// TIA Portal project "LearningFactory_4_0_24V_V00" (V16)

(* hardware
DEVICE "ET 200SP-Station_1"  ET 200SP-Station
   slot 0: "Baugruppenträger_0"  Rack  6ES5 710-8MAx1
   slot 1: "PLC"  CPU 1512SP-1 PN  6ES7 512-1DK01-0AB0  V2.6
   slot 2: "DO1+2"  DQ 16x24VDC/0.5A ST  6ES7 132-6BH01-0BA0  V0.0
      slot 1: "DO1+2"  DQ 16x24VDC/0.5A ST
   slot 3: "DO3+4"  DQ 16x24VDC/0.5A ST  6ES7 132-6BH01-0BA0  V0.0
      slot 1: "DO3+4"  DQ 16x24VDC/0.5A ST
   slot 4: "DO5+6"  DQ 16x24VDC/0.5A ST  6ES7 132-6BH01-0BA0  V0.0
      slot 1: "DO5+6"  DQ 16x24VDC/0.5A ST
   slot 5: "DO7-14"  DQ 4x24VDC/2A HS  6ES7 132-6BD20-0DA0  V2.0
      slot 1: "DO7-14"  DQ 4x24VDC/2A HS
   slot 6: "DO15-22"  DQ 4x24VDC/2A HS  6ES7 132-6BD20-0DA0  V2.0
      slot 1: "DO15-22"  DQ 4x24VDC/2A HS
   slot 7: "DO23-30"  DQ 4x24VDC/2A HS  6ES7 132-6BD20-0DA0  V2.0
      slot 1: "DO23-30"  DQ 4x24VDC/2A HS
   slot 8: "DI1+2"  DI 16x24VDC ST  6ES7 131-6BH01-0BA0  V0.0
      slot 1: "DI1+2"  DI 16x24VDC ST
   slot 9: "DI3+4"  DI 16x24VDC ST  6ES7 131-6BH01-0BA0  V0.0
      slot 1: "DI3+4"  DI 16x24VDC ST
   slot 10: "DI5"  DI 8x24VDC HS  6ES7 131-6BF00-0DA0  V1.0
      slot 1: "DI5"  DI 8x24VDC HS
   slot 11: "DI6"  DI 8x24VDC HS  6ES7 131-6BF00-0DA0  V1.0
      slot 1: "DI6"  DI 8x24VDC HS
   slot 12: "AI7-10"  AI 2xU ST  6ES7 134-6FB00-0BA1  V1.0
      slot 1: "AI7-10"  AI 2xU ST
   slot 13: "End"  Server module  6ES7 193-6PA00-0AA0  V1.1
      slot 1: "End"  Server module
   slot 127: "BA 2xRJ45"  BA 2xRJ45  6ES7 193-6AR00-0AA0  V0.0
      slot 32769: "Port_1"  6ES7 193-6AR00-0AA0
      slot 32770: "Port_2"  6ES7 193-6AR00-0AA0
*)

// ===== PLC "PLC"  CPU 1512SP-1 PN =====

VAR_GLOBAL   // PLC tag table "VGR - Vacuum Gripper Robot"
   "IX_VGR_RefSwitchVerticalAxis_I1" AT %I1.6 : Bool;   // VGR - I1 = Reference switch vertical axis
   "IX_VGR_RefSwitchHorizontalAxis_I2" AT %I3.6 : Bool;   // VGR - I2 = Reference switch horizontal axis
   "IX_VGR_RefSwitchRotate_I3" AT %I3.7 : Bool;   // VGR - I3 = Reference switch rotate
   "IX_VGR_EncoderVerticalAxisImp1_B1" AT %I6.0 : Bool;   // VGR - B1 = Encoder vertical axis imulse 1
   "IX_VGR_EncoderVerticalAxisImp2_B2" AT %I6.4 : Bool;   // VGR - B2 = Encoder vertical axis imulse 2
   "IX_VGR_EncoderHorizontalAxisImp1_B3" AT %I6.1 : Bool;   // VGR - B3 = Encoder horizontal axis imulse 1
   "IX_VGR_EncoderHorizontalAxisImp2_B4" AT %I6.5 : Bool;   // VGR - B4 = Encoder horizontal axis imulse 2
   "IX_VGR_EncoderRotateImp1_B5" AT %I6.2 : Bool;   // VGR - B5 = Encoder rotate impulse 1
   "IX_VGR_EncoderRotateImp2_B6" AT %I6.6 : Bool;   // VGR - B6 = Encoder rotate impulse 2
   "QX_VGR_M1_VerticalAxisUp_Q1" AT %Q2.0 : Bool;   // VGR - Q1 = Motor M1 vertical axis up
   "QX_VGR_M1_VerticalAxisDown_Q2" AT %Q2.1 : Bool;   // VGR - Q2 = Motor M1 vertical axis down
   "QX_VGR_M2_HorizontalAxisBackward_Q3" AT %Q2.2 : Bool;   // VGR - Q3 = Motor M2 horizontal axis backward
   "QX_VGR_M2_HorizontalAxisForward_Q4" AT %Q2.3 : Bool;   // VGR - Q4 = Motor M2 horizontal axis forward
   "QX_VGR_M3_RotateClockwise_Q5" AT %Q2.4 : Bool;   // VGR - Q5 = Motor M3 rotate clockwise
   "QX_VGR_M3_RotateCounterclockwise_Q6" AT %Q2.5 : Bool;   // VGR - Q6 = Motor M3 rotate counterclockwise
   "QX_VGR_Compressor_Q7" AT %Q2.6 : Bool;   // VGR - Q7 = Compressor
   "QX_VGR_ValveVacuum_Q8" AT %Q2.7 : Bool;   // VGR - Q8 = Valve vacuum
   "QW_VGR_PWM_Vertical_M1" AT %QW15 : Int;   // VGR = PWM Motor M1 vertical axis
   "QW_VGR_PWM_Horizontal_M2" AT %QW17 : Int;   // VGR = PWM Motor M2 horizontal axis
   "QW_VGR_PWM_Rotate_M3" AT %QW19 : Int;   // VGR = PWM Motor M3 rotate axis
END_VAR

VAR_GLOBAL   // PLC tag table "HBW - Automated High-Bay Warehouse"
   "IX_HBW_RefSwitchHorizontalAxis_I1" AT %I1.0 : Bool;   // HBW - I1 = Reference switch horizontal axis
   "IX_HBW_LightBarrierInside_I2" AT %I1.1 : Bool;   // HBW - I2 = Light barrier inside
   "IX_HBW_LightBarrierOutside_I3" AT %I1.2 : Bool;   // HBW - I3 = Light barrier outside
   "IX_HBW_RefSwitchVerticalAxis_I4" AT %I1.3 : Bool;   // HBW - I4 = Reference switch vertical axis
   "IX_HBW_TrailSensor1Lower_A1" AT %I5.0 : Bool;   // HBW - A1 = Trail sensor (signal 1, lower)
   "IX_HBW_TrailSensor2Upper_A2" AT %I5.4 : Bool;   // HBW - A2 = Trail sensor (signal 2, upper)
   "IX_HBW_EncoderVerticalAxisImp1_B3" AT %I5.2 : Bool;   // HBW - B3 = Encoder vertical axis imulse 1
   "IX_HBW_EncoderVerticalAxisImp2_B4" AT %I5.6 : Bool;   // HBW - B4 = Encoder vertical axis imulse 2
   "IX_HBW_EncoderHorizontalAxisImp1_B1" AT %I5.1 : Bool;   // HBW - B1 = Encoder horizontal axis imulse 1
   "IX_HBW_EncoderHorizontalAxisImp2_B2" AT %I5.5 : Bool;   // HBW - B2 = Encoder horizontal axis imulse 2
   "IX_HBW_SwitchCantileverFront_I5" AT %I1.4 : Bool;   // HBW - I5 = Reference switch cantilever front
   "IX_HBW_SwitchCantileverBack_I6" AT %I1.5 : Bool;   // HBW - I6 = Reference switch cantilever back
   "QX_HBW_M1_ConveyorBeltForward_Q1" AT %Q1.0 : Bool;   // HBW - Q1 = Motor M1 conveyor belt forward
   "QX_HBW_M1_ConveyorBeltBackward_Q2" AT %Q1.1 : Bool;   // HBW - Q2 = Motor M1 conveyor belt backward
   "QX_HBW_M2_HorizontalTowardsRack_Q3" AT %Q1.2 : Bool;   // HBW - Q3 = Motor M2 horizontal towards rack
   "QX_HBW_M2_HorizontalTowardsConveyorBelt_Q4" AT %Q1.3 : Bool;   // HBW - Q4 = Motor M2 horizontal towards conveyor belt
   "QX_HBW_M3_VerticalAxisDownward_Q5" AT %Q1.4 : Bool;   // HBW - Q5 = Motor M3 vertical axis downward
   "QX_HBW_M3_VerticalAxisUpward_Q6" AT %Q1.5 : Bool;   // HBW - Q6 = Motor M3 vertical axis upward
   "QX_HBW_M4_CantileverForward_Q7" AT %Q1.6 : Bool;   // HBW - Q7 = Motor M4 cantilever forward
   "QX_HBW_M4_CantileverBackward_Q8" AT %Q1.7 : Bool;   // HBW - Q8 = Motor M4 cantilever backward
   "QW_HBW_PWM_ConveyorBelt_M1" AT %QW7 : Int;   // HBW = PWM Motor M1 conveyor belt
   "QW_HBW_PWM_HorizontalAxis_M2" AT %QW9 : Int;   // HBW = PWM Motor M2 horizontal axis
   "QW_HBW_PWM_VerticalAxis_M3" AT %QW11 : Int;   // HBW = PWM Motor M3 vertical axis
   "QW_HBW_PWM_Cantilever_M4" AT %QW13 : Int;   // HBW = PWM Motor M4 cantilever
END_VAR

VAR_GLOBAL   // PLC tag table "SLD - Sorting Line with Detection"
   "IX_SLD_PulseCounter_I1" AT %I3.0 : Bool;   // SLD - I1 = Pulse counter
   "IX_SLD_LightBarrierInlet_I2" AT %I3.1 : Bool;   // SLD - I2 = Light barrier inlet
   "IX_SLD_LightBarrierBehindColorSensor_I3" AT %I3.2 : Bool;   // SLD - I3 = Light barrier behind color sensor
   "IW_SLD_ColorSensor_A4" AT %IW7 : Word;   // SLD - A4 = Color sensor
   "IX_SLD_LightBarrierWhite_I5" AT %I3.3 : Bool;   // SLD - I5 = Light barrier white
   "IX_SLD_LightBarrierRed_I6" AT %I3.4 : Bool;   // SLD - I6 = Light barrier red
   "IX_SLD_LightBarrierBlue_I7" AT %I3.5 : Bool;   // SLD - I7 = Light barrier blue
   "QX_SLD_M1_ConveyorBelt_Q1" AT %Q5.0 : Bool;   // SLD - Q1 = Motor M1conveyor belt
   "QX_SLD_Compressor_Q2" AT %Q5.1 : Bool;   // SLD - Q2 = Compressor
   "QX_SLD_ValveFirstEjectorWhite_Q3" AT %Q5.2 : Bool;   // SLD - Q3 = Valve first ejector (white)
   "QX_SLD_ValveSecondEjectorRed_Q4" AT %Q5.3 : Bool;   // SLD - Q4 = Valve second ejector (red)
   "QX_SLD_ValveThirdEjectorBlue_Q5" AT %Q5.4 : Bool;   // SLD - Q5 = Valve third ejector (blue)
END_VAR

VAR_GLOBAL   // PLC tag table "MPO - Multi Processing Station with Oven"
   "IX_MPO_RefSwitchTurnTable_PosVac_I1" AT %I1.7 : Bool;   // MPO - I1 = Reference switch turn-table (position vacuum)
   "IX_MPO_RefSwitchTurnTable_PosBelt_I2" AT %I2.0 : Bool;   // MPO - I2 = Reference switch turn-table (position belt)
   "IX_MPO_LightBarrierEndOfConBelt_I3" AT %I2.1 : Bool;   // MPO - I3 = Light barrier end of conveyor belt
   "IX_MPO_RefSwitchTurnTable_PosSaw_I4" AT %I2.2 : Bool;   // MPO - I4 = Reference switch turn-table (position saw)
   "IX_MPO_RefSwitchVac_PosTurnTable_I5" AT %I2.3 : Bool;   // MPO - I5 = Reference switch vacuum (position turn-table)
   "IX_MPO_RefSwitchOvenFeederInside_I6" AT %I2.4 : Bool;   // MPO - I6 = Reference switch oven feeder inside
   "IX_MPO_RefSwitchOvenFeederOutside_I7" AT %I2.5 : Bool;   // MPO - I7 = Reference switch oven feeder outside
   "IX_MPO_RefSwitchVac_PosOven_I8" AT %I2.6 : Bool;   // MPO - I8 = Reference switch vacuum (position oven)
   "IX_MPO_LightBarrierOven_I9" AT %I2.7 : Bool;   // MPO - I9 = Light barrier oven
   "QX_MPO_M1_TurnTableClockwise_Q1" AT %Q3.0 : Bool;   // MPO - Q1 = Motor M1 turn-table clockwise
   "QX_MPO_M1_TurnTableCounterclockwise_Q2" AT %Q3.1 : Bool;   // MPO - Q2 = Motor M1 turn-table counterclockwise
   "QX_MPO_M2_ConveyorBeltForward_Q3" AT %Q3.2 : Bool;   // MPO - Q3 = Motor M2 conveyor belt forward
   "QX_MPO_M3_Saw_Q4" AT %Q3.3 : Bool;   // MPO - Q4 = Motor M3 saw
   "QX_MPO_M4_OvenFeederRetract_Q5" AT %Q3.4 : Bool;   // MPO - Q5 = Motor M4 oven feeder retract
   "QX_MPO_M4_OvenFeederExtend_Q6" AT %Q3.5 : Bool;   // MPO - Q6 = Motor M4 oven feeder extend
   "QX_MPO_M5_VacuumTowardsOven_Q7" AT %Q3.6 : Bool;   // MPO - Q7 = Motor M5 vacuum towards oven
   "QX_MPO_M5_VacuumTowardsTurnTable_Q8" AT %Q3.7 : Bool;   // MPO - Q8 = Motor M5 vacuum towards turn-table
   "QX_MPO_LightOven_Q9" AT %Q4.0 : Bool;   // MPO - Q9 = Light oven
   "QX_MPO_Compressor_Q10" AT %Q4.1 : Bool;   // MPO - Q10 = Compressor
   "QX_MPO_ValveVacuum_Q11" AT %Q4.2 : Bool;   // MPO - Q11 = Valve vacuum
   "QX_MPO_ValveLowering_Q12" AT %Q4.3 : Bool;   // MPO - Q12 = Valve lowering
   "QX_MPO_ValveOvenDoor_Q13" AT %Q4.4 : Bool;   // MPO - Q13 = Valve oven door
   "QX_MPO_ValveFeeder_Q14" AT %Q4.5 : Bool;   // MPO - Q14 = Valve feeder
   "QW_MPO_PWM_TurnTable_M1" AT %QW23 : Int;   // MPO = PWM Motor M1 turn-table
   "QW_MPO_PWM_Vacuum_M5" AT %QW25 : Int;   // MPO = PWM Motor M5 turn-table
END_VAR

VAR_GLOBAL   // PLC tag table "SSC - Sensor-Station Camera"
   "IX_SSC_RefSwitchVerticalAxis_I1" AT %I4.0 : Bool;   // SSC - ?? = Reference switch vertical axis / SSC - I1 = Reference switch vertical axis
   "IX_SSC_RefSwitchHorizontalAxis_I2" AT %I4.1 : Bool;   // SSC - ?? = Reference switch horizontal axis / SSC - I2 = Reference switch horizontal axis
   "IX_SSC_LightBarrierStorage_I3" AT %I4.3 : Bool;   // SSC - ?? = Light barrier inlet / SSC - I3 = Light barrier inlet
   "IX_SSC_LightBarrierOutsourcing_I4" AT %I4.2 : Bool;   // SSC - ?? = Light barrier behind color sensor / SSC - I4 = Light barrier behind color sensor
   "IW_SSC_ColorSensor_A1" AT %IW9 : Word;   // SSC - ?? = Color sensor / SSC - A1 = Color sensor
   "IX_SSC_EncoderVerticalAxisImp1_B1" AT %I5.3 : Bool;   // SSC - ?? = Encoder vertical axis imulse 1 / SSC - B1 = Encoder vertical axis imulse 1
   "IX_SSC_EncoderVerticalAxisImp2_B2" AT %I5.7 : Bool;   // SSC - ?? = Encoder vertical axis imulse 2 / SSC - B2 = Encoder vertical axis imulse 2
   "IX_SSC_EncoderHorizontalAxisImp1_B3" AT %I6.3 : Bool;   // SSC - ?? = Encoder horizontal axis imulse 1 / SSC - B3 = Encoder horizontal axis imulse 1
   "IX_SSC_EncoderHorizontalAxisImp2_B4" AT %I6.7 : Bool;   // SSC - ?? = Encoder horizontal axis imulse 2 / SSC - B4 = Encoder horizontal axis imulse 2
   "QX_SSC_M1_VerticalAxisUp_Q1" AT %Q6.0 : Bool;   // SSC - ?? = Motor M1 vertical axis up / SSC - Q1 = Motor M1 vertical axis up
   "QX_SSC_M1_VerticalAxisDown_Q2" AT %Q6.1 : Bool;   // SSC - ?? = Motor M1 vertical axis down / SSC - Q2 = Motor M1 vertical axis down
   "QX_SSC_M2_HorizontalAxisClockwise_Q3" AT %Q6.3 : Bool;   // SSC - ?? = Motor M2 horizontal axis backward / SSC - Q3 = Motor M2 horizontal axis backward
   "QX_SSC_M2_HorizontalAxisCounterclockwise_Q4" AT %Q6.2 : Bool;   // SSC - ?? = Motor M2 horizontal axis forward / SSC - Q4 = Motor M2 horizontal axis forward
   "QX_SSC_LED_Green_Q5" AT %Q6.4 : Bool;   // SSC - ?? = / SSC - Q5 = LED Green
   "QX_SSC_LED_Yellow_Q6" AT %Q6.5 : Bool;   // SSC - ?? = / SSC - Q6 = LED Yellow
   "QX_SSC_LED_Red_Q7" AT %Q6.6 : Bool;   // SSC - ?? = / SSC - Q7 = LED Red
   "QX_SSC_LED_Red_Online_Q8" AT %Q6.7 : Bool;   // SSC - ?? = / SSC - Q8 = LED Red Online
   "QW_SSC_PWM_Vertical_M1" AT %QW27 : Int;   // SSC - ?? = / SSC = PWM Motor M1 vertical axis
   "QW_SSC_PWM_Horizontal_M2" AT %QW29 : Int;   // SSC - ?? = / SSC = PWM Motor M2 horizontal axis
END_VAR

TYPE "typ_VGR"
   STRUCT
      x_NFC_Start_First : Bool;
      x_NFC_Start : Bool;
      x_NFC_Completed : Bool;
      x_HBW_Storage : Bool;
      x_HBW_Outsource : Bool;
      s_HBW_Outsource_Typ : String;
      x_HBW_Discards : Bool;
      x_HBW_PickedUp : Bool;
      x_MPO_Req_Discard : Bool;
      x_MPO_Discards : Bool;
      x_Ready_For_Outsource : Bool;
      x_State_Process : Bool;
      x_Workpiece_NiO : Bool;
      horizontal_Axis : "typ_Axis";
      vertical_Axis : "typ_Axis";
      rotate_Axis : "typ_Axis";
      Workpiece : "typ_Workpiece";
      History : Array[1..20] of "typ_History";
      di_Pos_DSI_horizontal : DInt;
      di_Pos_DSI_Collect_vertical : DInt;
      di_Pos_DSI_Discard_vertical : DInt;
      di_Offset_Pos_DSI_NFC_vertical : DInt;
      di_Pos_DSI_rotate : DInt;
      di_Pos_DSO_horizontal : DInt;
      di_Pos_DSO_Collect_vertical : DInt;
      di_Pos_DSO_Discard_vertical : DInt;
      di_Offset_Pos_DSO_vertical : DInt;
      di_Pos_DSO_rotate : DInt;
      di_Pos_Color_horizontal : DInt;
      di_Pos_Color_vertical : DInt;
      di_Pos_Color_rotate : DInt;
      di_Pos_NFC_horizontal : DInt;
      di_Pos_NFC_vertical : DInt;
      di_Pos_NFC_rotate : DInt;
      di_Pos_MPO_horizontal : DInt;
      di_Pos_MPO_vertical : DInt;
      di_Offset_Pos_MPO_vertical : DInt;
      di_Pos_MPO_rotate : DInt;
      di_Pos_HBW_horizontal : DInt;
      di_Offset_Pos_HBW_horizontal : DInt;
      di_Pos_HBW_Collect_vertical : DInt;
      di_Pos_HBW_Discard_vertical : DInt;
      di_Offset_Pos_HBW_vertical : DInt;
      di_Pos_HBW_rotate : DInt;
      di_Pos_NiO_horizontal : DInt;
      di_Pos_NiO_vertical : DInt;
      di_Pos_NiO_rotate : DInt;
      di_Pos_SLD_Blue_horizontal : DInt;
      di_Pos_SLD_Blue_vertical : DInt;
      di_Pos_SLD_Blue_rotate : DInt;
      di_Pos_SLD_Red_horizontal : DInt;
      di_Pos_SLD_Red_vertical : DInt;
      di_Pos_SLD_Red_rotate : DInt;
      di_Pos_SLD_White_horizontal : DInt;
      di_Pos_SLD_White_vertical : DInt;
      di_Pos_SLD_White_rotate : DInt;
   END_STRUCT;
END_TYPE

TYPE "typ_SetupAxis"
   STRUCT
      x_Setup_Activ : Bool;   // Einrichten Kalibrieren aktiv / Set up calibration active
      i_AxisSelection : Int;   // Nummer der Achse / Number of the axis
      i_Function : Int;   // 0= Automatic, 10=Ref. Fahrt, 20= Tippen, 30=Tippen mit Schritweite, 40= Pos. Anfahren / 0 = automatic, 10 = ref. Travel, 20 = tap, 30 = tap with step width, 40 = start
      x_Set_Ref_Pos : Bool;   // Referenzwert setzen / Set reference value
      x_Set_Soft_End_Pos : Bool;   // Softwareendlagen setzen / Set software end positions
      x_Approach_Ref_Pos : Bool;   // Referenz anfahren / Approach reference
      x_Axis_Pos : Bool;   // Achse positiv / Axis positiv
      x_Axis_Neg : Bool;   // Achse negativ / Axis negative
      x_Approach_Target_Pos : Bool;   // Zielposition anfahren / Approach Target position
      w_Increment : Word;   // Inkremente pro Schritt / Increments per step
      i_PWM : Int;   // PWM Signal
      di_Target_Position : DInt;   // Zielposition / Target position
      di_ActualPosition : DInt;   // Aktuelle Position / Actual position
      di_Ref_Pos : DInt;   // Referenzposition / Reference position
      di_Actual_Ref_Pos : DInt;   // Aktuelle Referenzposition / Current reference position
      di_Soft_End_Pos_Neg : DInt;   // Softwareendlage negativ / Software end position negative
      di_Actual_Soft_End_Pos_Neg : DInt;   // Aktuelle Softwareendlage negativ / Current software end position negative
      di_Soft_End_Pos_Pos : DInt;   // Softwareendlage positiv / Software end position positiv
      di_Actual_Soft_End_Pos_Pos : DInt;   // Aktuelle Softwareendlage positiv / Current software end position positiv
      di_LoopValue : DInt;   // Schleifenwert / Loop value
   END_STRUCT;
END_TYPE

TYPE "typ_Axis_Data"
   STRUCT
      di_Pos_Soft_Switch : DInt := 0;
      di_Neg_Soft_Switch : DInt := 0;
      di_Ref_Pos : DInt := 0;
      di_Loop_Value : DInt := 0;
      di_Pos_Window : DInt := 15;
   END_STRUCT;
END_TYPE

TYPE "typ_Axis"
   STRUCT
      x_Start_Positioning : Bool;
      x_Reference : Bool;
      x_Referenced : Bool;
      x_Position_Reached : Bool;
      di_Target_Position : DInt;
      di_Increment : DInt;
      di_Actual_Position : DInt := 0;
      i_PWM : Int;
      Config : "typ_Axis_Data";
   END_STRUCT;
END_TYPE

TYPE "typ_SSC"
   STRUCT
      x_Error : Bool;
      di_Pos_Centre_Horizontal : DInt;
      di_Pos_Centre_Vertical : DInt;
      di_Pos_HBW_Horizontal : DInt;
      di_Pos_HBW_Vertical : DInt;
      w_Threshold_White_Red : Word;
      w_Threshold_Red_Blue : Word;
      Horizontal_Axis : "typ_Axis";
      Vertical_Axis : "typ_Axis";
      Workpiece : "typ_Workpiece";
      History : Array[1..20] of "typ_History";
   END_STRUCT;
END_TYPE

TYPE "typ_HBW"
   STRUCT
      x_HBW_PickedUp_Accepted : Bool;
      x_HBW_Discards_Accepted : Bool;
      x_HBW_PickUp_Ready : Bool;
      x_HBW_Container_Available : Bool;
      x_Error : Bool;
      di_PosBelt_Horizontal : DInt;
      di_PosBelt_Vertical : DInt;
      di_Offset_Pos_Belt_Vertical : DInt;
      di_PosRack_A1_Horizontal : DInt;
      di_PosRack_A1_Vertical : DInt;
      di_PosRack_B2_Horizontal : DInt;
      di_PosRack_B2_Vertical : DInt;
      di_PosRack_C3_Horizontal : DInt;
      di_PosRack_C3_Vertical : DInt;
      di_Offset_Pos_Rack_Vertical : DInt;
      i_PWM_ConveyorBelt : Int := 800;
      i_PWM_Cantilever : Int := 800;
      Workpiece : "typ_Workpiece";
      History : Array[1..20] of "typ_History";
      Rack_Pos : Array[1..3, 1..3] of "typ_Rack_Pos";
      Rack_Workpiece : Array[1..3, 1..3] of "typ_Workpiece";
      Rack_History : Array[1..3, 1..3] of "typ_Rack_History";
      Horizontal_Axis : "typ_Axis";
      Vertical_Axis : "typ_Axis";
   END_STRUCT;
END_TYPE

TYPE "typ_Rack_Pos"
   STRUCT
      di_PosRack_Horizontal : DInt;
      di_PosRack_Vertical : DInt;
   END_STRUCT;
END_TYPE

TYPE "typ_MPO"
   STRUCT
      x_Discard_Ready : Bool;
      x_MPO_Discards_Accepted : Bool;
      x_Error : Bool;
      i_PWM_TurnTable : Int := 700;
      i_PWM_Vacuum : Int := 1000;
      Workpiece : "typ_Workpiece";
      History : Array[1..20] of "typ_History";
   END_STRUCT;
END_TYPE

TYPE "typ_SLD"
   STRUCT
      x_Error : Bool;
      i_CounterValue_Blue : Int := 8;
      i_CounterValue_White : Int := 2;
      i_CounterValue_Red : Int := 4;
      i_Counter_Actual : Int;
      w_Threshold_White_Red : Word;
      w_Threshold_Red_Blue : Word;
      Workpiece : "typ_Workpiece";
      History : Array[1..20] of "typ_History";
   END_STRUCT;
END_TYPE

TYPE "typ_Setup"
   STRUCT
      x_Clean_Rack_HBW : Bool;
      x_AcknowledgeButton : Bool;
      x_Color_Sensor_Calibration : Bool;
      x_Set_Calib_Value_Color_Blue : Bool;
      x_Set_Calib_Value_Color_White : Bool;
      x_Set_Calib_Value_Color_Red : Bool;
      x_Calculate_Value_Color : Bool;
      i_Color_Sensor_Selection : Int;
      w_Calib_ColorValue_Blue : Word;
      w_Calib_ColorValue_White : Word;
      w_Calib_ColorValue_Red : Word;
      w_Threshold_White_Red : Word;
      w_Threshold_Red_Blue : Word;
      w_Actual_ColorValue : Word;
      x_Set_Pos_Activ : Bool;   // Einrichten Kalibrieren aktiv / Set up calibration active
      x_Start_Positioning : Bool;
      x_Final_Positioning : Bool;
      x_Home_Positioning : Bool;
      x_Start_Offset : Bool;
      i_Pos_Selection : Int;   // Nummer der Achse / Number of the axis
      di_Pos_Horizontal : DInt;
      di_Pos_Vertical : DInt;
      di_Pos_Rotate : DInt;
      x_Counter_Value_Calibration : Bool;   // Einrichten Kalibrieren aktiv
      i_Calib_CounterValue_Blue : Int := 26;
      i_Calib_CounterValue_White : Int := 5;
      i_Calib_CounterValue_Red : Int := 16;
      x_Set_CounterValues : Bool;   // Einrichten Kalibrieren aktiv
      x_Activate_Continuous_Operation : Bool;
   END_STRUCT;
END_TYPE

TYPE "typ_Rack_History"
   STRUCT
      History : Array[1..20] of "typ_History";
   END_STRUCT;
END_TYPE

// folder: Dashboard types

TYPE "typ_Stock_Item"
   STRUCT
      ldt_ts : LDT;
      StockItem : Array[1..3, 1..3] of "typ_Workpiece";
      s_location : String;
   END_STRUCT;
END_TYPE

TYPE "typ_Acknowledgment_Client"
   STRUCT
      ldt_ts : LDT;
      i_code : Int;
      Workpiece : "typ_Workpiece";
   END_STRUCT;
END_TYPE

TYPE "typ_State_Client"
   STRUCT
      ldt_ts : LDT;
      s_station : String;
      i_code : Int;
      s_description : String;
      x_active : Bool;
      s_target : String;
   END_STRUCT;
END_TYPE

TYPE "typ_Broadcast"
   STRUCT
      ldt_ts : LDT;
      di_hardwareId : DInt;
      di_hardwareModel : DInt;
      s_softwareName : String;
      di_softwareVersion : DInt;
      s_message : String;
   END_STRUCT;
END_TYPE

TYPE "typ_Config_Camera_Picture"
   STRUCT
      ldt_ts : LDT;
      di_period : DInt;
   END_STRUCT;
END_TYPE

TYPE "typ_Config_Brightness_Sensor"
   STRUCT
      ldt_ts : LDT;
      x_on : Bool;
      i_fps : Int;
   END_STRUCT;
END_TYPE

TYPE "typ_Config_Enviorment_Sensor"
   STRUCT
      ldt_ts : LDT;
      di_period : DInt;
   END_STRUCT;
END_TYPE

TYPE "typ_History"
   STRUCT
      ldt_ts : LDT;
      i_code : Int;
   END_STRUCT;
END_TYPE

TYPE "typ_Pos_Pan_Tilt_Unit_Mov"
   STRUCT
      ldt_ts : LDT;
      s_cmd : String;
      i_degree : Int;
   END_STRUCT;
END_TYPE

TYPE "typ_Workpiece"
   STRUCT
      s_id : String;
      s_type : String;
      s_state : String;
   END_STRUCT;
END_TYPE

TYPE "typ_Order_Workpiece_Buttons_State"
   STRUCT
      ldt_ts : LDT;
      s_state : String;
      s_type : String;
   END_STRUCT;
END_TYPE

TYPE "typ_NFC_Module_State"
   STRUCT
      ldt_ts : LDT;
      Workpiece : "typ_Workpiece";
      History : Array[1..20] of "typ_History";
   END_STRUCT;
END_TYPE

TYPE "typ_VGR_Trigger"
   STRUCT
      ldt_ts : LDT;
      i_code : Int;
      Workpiece : "typ_Workpiece";
   END_STRUCT;
END_TYPE

TYPE "typ_Alert_Message"
   STRUCT
      ldt_ts : LDT;
      s_id : String;
      s_data : String;
      i_code : Int;
   END_STRUCT;
END_TYPE

TYPE "typ_Camera_Picture"
   STRUCT
      ldt_ts : LDT;
      s_data : String;
   END_STRUCT;
END_TYPE

TYPE "typ_Pos_Pan_Tilt_Unit_Enc"
   STRUCT
      ldt_ts : LDT;
      r_pan : Real;
      r_tilt : Real;
   END_STRUCT;
END_TYPE

TYPE "typ_Brightness_Sensor"
   STRUCT
      ldt_ts : LDT;
      r_br : Real;
      i_ldr : Int;
   END_STRUCT;
END_TYPE

TYPE "typ_Environment_Sensor"
   STRUCT
      ldt_ts : LDT;
      r_t : Real;
      r_rt : Real;
      r_h : Real;
      r_rh : Real;
      r_p : Real;
      i_iaq : Int;
      i_aq : Int;
      di_gr : DInt;
   END_STRUCT;
END_TYPE

TYPE "typ_Order_Workpiece_Buttons"
   STRUCT
      ldt_ts : LDT;
      s_type : String;
   END_STRUCT;
END_TYPE

TYPE "typ_Action_Buttons_NFC_Module"
   STRUCT
      ldt_ts : LDT;
      s_cmd : String;
   END_STRUCT;
END_TYPE

TYPE "typ_Joysticks"
   STRUCT
      ldt_ts : LDT;
      r_br : Real;
      i_ldr : Int;
   END_STRUCT;
END_TYPE

// folder: Interface Dashboard

TYPE "typ_MQTT_Interface_Dashboard"
   STRUCT
      Subscribe : "typ_MQTT_Interface_Dashboard_Subscribe";
      Publish : "typ_MQTT_ Interface_Dashboard_Publish";
   END_STRUCT;
END_TYPE

TYPE "typ_MQTT_ Interface_Dashboard_Publish"
   STRUCT
      ldt_AcknowledgeButton : LDT;
      ConfigRateEnviormentSensor : "typ_Config_Enviorment_Sensor";
      ConfigRateBrightnessSensor : "typ_Config_Brightness_Sensor";
      ConfigRateCameraPicture : "typ_Config_Camera_Picture";
      PosPanTiltUnit : "typ_Pos_Pan_Tilt_Unit_Mov";
      OrderWorkpieceButton : "typ_Order_Workpiece_Buttons";
      ActionButtonNFCModule : "typ_Action_Buttons_NFC_Module";
   END_STRUCT;
END_TYPE

TYPE "typ_MQTT_Interface_Dashboard_Subscribe"
   STRUCT
      EnvironmentSensor : "typ_Environment_Sensor";
      BrightnessSensor : "typ_Brightness_Sensor";
      CameraPicture : "typ_Camera_Picture";
      PosPanTiltUnit : "typ_Pos_Pan_Tilt_Unit_Enc";
      AlertMessage : "typ_Alert_Message";
      Broadcast : "typ_Broadcast";
      State_HBW : "typ_State_Client";
      State_VGR : "typ_State_Client";
      State_MPO : "typ_State_Client";
      State_SLD : "typ_State_Client";
      State_DSI : "typ_State_Client";
      State_DSO : "typ_State_Client";
      Stock_HBW : "typ_Stock_Item";
      State_Order : "typ_Order_Workpiece_Buttons_State";
      State_NFC_Device : "typ_NFC_Module_State";
   END_STRUCT;
END_TYPE

// folder: Interface TXT Controller

TYPE "typ_MQTT_Interface_TXT_Controller"
   STRUCT
      Subscribe : "typ_MQTT_Interface_TXT_Controler_Subscribe";
      Publish : "typ_MQTT_ Interface_TXT_Controler_Publish";
   END_STRUCT;
END_TYPE

TYPE "typ_MQTT_ Interface_TXT_Controler_Publish"
   STRUCT
      ActionButtonNFCModule : "typ_SPS_Action_Buttons_NFC_Module";
   END_STRUCT;
END_TYPE

TYPE "typ_MQTT_Interface_TXT_Controler_Subscribe"
   STRUCT
      State_NFC_Device : "typ_SPS_NFC_Module_State";
   END_STRUCT;
END_TYPE

// folder: TXT Controler Types

TYPE "typ_SPS_NFC_Module_State"
   STRUCT
      ldt_ts : LDT;
      Workpiece : "typ_Workpiece";
      History : Array[1..20] of "typ_History";
   END_STRUCT;
END_TYPE

TYPE "typ_SPS_Action_Buttons_NFC_Module"
   STRUCT
      ldt_ts : LDT;
      s_cmd : String;
      Workpiece : "typ_Workpiece";
      History : Array[1..20] of "typ_History";
   END_STRUCT;
END_TYPE

// folder: 2. Cloud

DATA_BLOCK "PRG_NFC_DB"   // DB12
{ S7_Optimized_Access := 'TRUE' }
VERSION : 0.1
// stored: InstanceOfName PRG_NFC
"PRG_NFC"
BEGIN
END_DATA_BLOCK

DATA_BLOCK "PRG_Acknowledge_DB"   // DB21
{ S7_Optimized_Access := 'TRUE' }
VERSION : 0.1
// stored: InstanceOfName PRG_Acknowledge
"PRG_Acknowledge"
BEGIN
END_DATA_BLOCK

DATA_BLOCK "PRG_Order_DB"   // DB25
{ S7_Optimized_Access := 'TRUE' }
VERSION : 0.1
// stored: InstanceOfName PRG_Order
"PRG_Order"
BEGIN
END_DATA_BLOCK

// folder: 3.1. VGR

DATA_BLOCK "PRG_VGR_Axis_horizontal_DB"   // DB8
{ S7_Optimized_Access := 'TRUE' }
VERSION : 0.1
// stored: InstanceOfName PRG_VGR_Axis_horizontal
"PRG_VGR_Axis_horizontal"
BEGIN
END_DATA_BLOCK

DATA_BLOCK "PRG_VGR_Axis_vertical_DB"   // DB9
{ S7_Optimized_Access := 'TRUE' }
VERSION : 0.1
// stored: InstanceOfName PRG_VGR_Axis_vertical
"PRG_VGR_Axis_vertical"
BEGIN
END_DATA_BLOCK

DATA_BLOCK "PRG_VGR_Axis_rotate_DB"   // DB10
{ S7_Optimized_Access := 'TRUE' }
VERSION : 0.1
// stored: InstanceOfName PRG_VGR_Axis_rotate
"PRG_VGR_Axis_rotate"
BEGIN
END_DATA_BLOCK

DATA_BLOCK "PRG_VGR_Axis_horizontal_Act_Pos_DB"   // DB15
{ S7_Optimized_Access := 'TRUE' }
VERSION : 0.1
// stored: InstanceOfName PRG_VGR_Axis_horizontal_Act_Pos
"PRG_VGR_Axis_horizontal_Act_Pos"
BEGIN
END_DATA_BLOCK

DATA_BLOCK "PRG_VGR_Ablauf_DB"   // DB19
{ S7_Optimized_Access := 'TRUE' }
VERSION : 0.1
// stored: InstanceOfName PRG_VGR_Ablauf
"PRG_VGR_Ablauf"
BEGIN
END_DATA_BLOCK

DATA_BLOCK "PRG_VGR_Axis_vertical_Act_Pos_DB"   // DB29
{ S7_Optimized_Access := 'TRUE' }
VERSION : 0.1
// stored: InstanceOfName PRG_VGR_Axis_vertical_Act_Pos
"PRG_VGR_Axis_vertical_Act_Pos"
BEGIN
END_DATA_BLOCK

DATA_BLOCK "PRG_VGR_Axis_rotate_Act_Pos_DB"   // DB31
{ S7_Optimized_Access := 'TRUE' }
VERSION : 0.1
// stored: InstanceOfName PRG_VGR_Axis_rotate_Act_Pos
"PRG_VGR_Axis_rotate_Act_Pos"
BEGIN
END_DATA_BLOCK

DATA_BLOCK "PRG_VGR_Set_Positioning_DB"   // DB34
{ S7_Optimized_Access := 'TRUE' }
VERSION : 0.1
// stored: InstanceOfName PRG_VGR_Set_Positioning
"PRG_VGR_Set_Positioning"
BEGIN
END_DATA_BLOCK

// folder: 3.2. HBW

DATA_BLOCK "PRG_HBW_Axis_Vertical_DB"   // DB14
{ S7_Optimized_Access := 'TRUE' }
VERSION : 0.1
// stored: InstanceOfName PRG_HBW_Axis_Vertical
"PRG_HBW_Axis_Vertical"
BEGIN
END_DATA_BLOCK

DATA_BLOCK "PRG_HBW_Axis_Horizontal_DB"   // DB18
{ S7_Optimized_Access := 'TRUE' }
VERSION : 0.1
// stored: InstanceOfName PRG_HBW_Axis_Horizontal
"PRG_HBW_Axis_Horizontal"
BEGIN
END_DATA_BLOCK

DATA_BLOCK "PRG_HBW_Ablauf_DB"   // DB22
{ S7_Optimized_Access := 'TRUE' }
VERSION : 0.1
// stored: InstanceOfName PRG_HBW_Ablauf
"PRG_HBW_Ablauf"
BEGIN
END_DATA_BLOCK

DATA_BLOCK "PRG_HBW_Axis_Horizontal_Act_Pos_DB"   // DB27
{ S7_Optimized_Access := 'TRUE' }
VERSION : 0.1
// stored: InstanceOfName PRG_HBW_Axis_Horizontal_Act_Pos
"PRG_HBW_Axis_Horizontal_Act_Pos"
BEGIN
END_DATA_BLOCK

DATA_BLOCK "PRG_HBW_Axis_Vertical_Act_Pos_DB"   // DB28
{ S7_Optimized_Access := 'TRUE' }
VERSION : 0.1
// stored: InstanceOfName PRG_HBW_Axis_Vertical_Act_Pos
"PRG_HBW_Axis_Vertical_Act_Pos"
BEGIN
END_DATA_BLOCK

DATA_BLOCK "PRG_HBW_Set_Positioning_DB"   // DB35
{ S7_Optimized_Access := 'TRUE' }
VERSION : 0.1
// stored: InstanceOfName PRG_HBW_Set_Positioning
"PRG_HBW_Set_Positioning"
BEGIN
END_DATA_BLOCK

// folder: 3.3. MPO

DATA_BLOCK "PRG_MPO_Ablauf_DB"   // DB5
{ S7_Optimized_Access := 'TRUE' }
VERSION : 0.1
// stored: InstanceOfName PRG_MPO_Ablauf
"PRG_MPO_Ablauf"
BEGIN
END_DATA_BLOCK

// folder: 3.4. SLD

DATA_BLOCK "PRG_SLD_Ablauf_DB"   // DB20
{ S7_Optimized_Access := 'TRUE' }
VERSION : 0.1
// stored: InstanceOfName PRG_SLD_Ablauf
"PRG_SLD_Ablauf"
BEGIN
END_DATA_BLOCK

DATA_BLOCK "PRG_SLD_Calibration_Color_DB"   // DB38
{ S7_Optimized_Access := 'TRUE' }
VERSION : 0.1
// stored: InstanceOfName PRG_SLD_Calibration_Color
"PRG_SLD_Calibration_Color"
BEGIN
END_DATA_BLOCK

DATA_BLOCK "PRG_SLD_Set_Counter_Values_DB"   // DB39
{ S7_Optimized_Access := 'TRUE' }
VERSION : 0.1
// stored: InstanceOfName PRG_SLD_Set_Counter_Values
"PRG_SLD_Set_Counter_Values"
BEGIN
END_DATA_BLOCK

// folder: 3.5. SSC

DATA_BLOCK "PRG_SSC_Axis_Vertical_DB"   // DB3
{ S7_Optimized_Access := 'TRUE' }
VERSION : 0.1
// stored: InstanceOfName PRG_SSC_Axis_Vertical
"PRG_SSC_Axis_Vertical"
BEGIN
END_DATA_BLOCK

DATA_BLOCK "PRG_SSC_Axis_Vertical_Act_Pos_DB"   // DB6
{ S7_Optimized_Access := 'TRUE' }
VERSION : 0.1
// stored: InstanceOfName PRG_SSC_Axis_Vertical_Act_Pos
"PRG_SSC_Axis_Vertical_Act_Pos"
BEGIN
END_DATA_BLOCK

DATA_BLOCK "PRG_SSC_Axis_Horizontal_DB"   // DB7
{ S7_Optimized_Access := 'TRUE' }
VERSION : 0.1
// stored: InstanceOfName PRG_SSC_Axis_Horizontal
"PRG_SSC_Axis_Horizontal"
BEGIN
END_DATA_BLOCK

DATA_BLOCK "PRG_SSC_Ablauf_DB"   // DB16
{ S7_Optimized_Access := 'TRUE' }
VERSION : 0.1
// stored: InstanceOfName PRG_SSC_Ablauf
"PRG_SSC_Ablauf"
BEGIN
END_DATA_BLOCK

DATA_BLOCK "PRG_SSC_Light_DB"   // DB26
{ S7_Optimized_Access := 'TRUE' }
VERSION : 0.1
// stored: InstanceOfName PRG_SSC_Light
"PRG_SSC_Light"
BEGIN
END_DATA_BLOCK

DATA_BLOCK "PRG_SSC_Axis_Horizontal_Act_Pos_DB"   // DB30
{ S7_Optimized_Access := 'TRUE' }
VERSION : 0.1
// stored: InstanceOfName PRG_SSC_Axis_Horizontal_Act_Pos
"PRG_SSC_Axis_Horizontal_Act_Pos"
BEGIN
END_DATA_BLOCK

DATA_BLOCK "PRG_DSI_Status_DB"   // DB32
{ S7_Optimized_Access := 'TRUE' }
VERSION : 0.1
// stored: InstanceOfName PRG_DSI_Status
"PRG_DSI_Status"
BEGIN
END_DATA_BLOCK

DATA_BLOCK "PRG_DSO_Status_DB"   // DB33
{ S7_Optimized_Access := 'TRUE' }
VERSION : 0.1
// stored: InstanceOfName PRG_DSO_Status
"PRG_DSO_Status"
BEGIN
END_DATA_BLOCK

DATA_BLOCK "PRG_SSC_Set_Positioning_DB"   // DB36
{ S7_Optimized_Access := 'TRUE' }
VERSION : 0.1
// stored: InstanceOfName PRG_SSC_Set_Positioning
"PRG_SSC_Set_Positioning"
BEGIN
END_DATA_BLOCK

DATA_BLOCK "PRG_SSC_Calibration_Color_DB"   // DB37
{ S7_Optimized_Access := 'TRUE' }
VERSION : 0.1
// stored: InstanceOfName PRG_SSC_Calibration_Color
"PRG_SSC_Calibration_Color"
BEGIN
END_DATA_BLOCK

// folder: 4. Global Declaration

DATA_BLOCK "gtyp_Interface_Dashboard"   // DB1
TITLE = Global Interface Dashboard Cloud
{ S7_Optimized_Access := 'TRUE' }
AUTHOR : A.Schaefer
VERSION : 0.0
BEGIN
END_DATA_BLOCK

DATA_BLOCK "gtyp_VGR"   // DB2
TITLE = Global DB VGR
{ S7_Optimized_Access := 'TRUE' }
AUTHOR : A.Schaefer
VERSION : 0.0
BEGIN
   di_Pos_DSI_Collect_vertical := 2950;
   di_Pos_MPO_vertical := 1800;
   di_Pos_HBW_Discard_vertical := 200;
   vertical_Axis.Config.di_Pos_Soft_Switch := 20000;
   horizontal_Axis.Config.di_Pos_Soft_Switch := 20000;
   rotate_Axis.Config.di_Pos_Soft_Switch := 20000;
   di_Pos_DSI_horizontal := 20;
   di_Pos_DSI_rotate := 30;
   di_Pos_Color_horizontal := 150;
   di_Pos_Color_rotate := 430;
   di_Pos_Color_vertical := 2450;
   di_Pos_NFC_vertical := 2450;
   di_Pos_NFC_horizontal := 900;
   di_Pos_NFC_rotate := 700;
   di_Pos_HBW_rotate := 5350;
   di_Offset_Pos_DSI_NFC_vertical := 1200;
   di_Offset_Pos_HBW_vertical := 100;
   di_Pos_HBW_horizontal := 600;
   di_Pos_SLD_Red_rotate := 1460;
   di_Pos_SLD_White_rotate := 1770;
   di_Pos_SLD_Blue_rotate := 1200;
   di_Pos_SLD_Red_vertical := 3100;
   di_Pos_SLD_White_vertical := 3100;
   di_Pos_SLD_Blue_vertical := 3100;
   di_Pos_SLD_Red_horizontal := 1580;
   di_Pos_SLD_White_horizontal := 1370;
   di_Pos_SLD_Blue_horizontal := 2150;
   di_Pos_DSO_rotate := 970;
   di_Pos_MPO_rotate := 3500;
   di_Pos_NiO_rotate := 1100;
   di_Pos_DSO_horizontal := 2070;
   di_Pos_DSO_Discard_vertical := 1480;
   di_Pos_NiO_vertical := 2700;
   di_Pos_MPO_horizontal := 3400;
   di_Pos_HBW_Collect_vertical := 650;
   di_Offset_Pos_MPO_vertical := 650;
   horizontal_Axis.i_PWM := 500;
   vertical_Axis.i_PWM := 500;
   rotate_Axis.i_PWM := 500;
   di_Offset_Pos_DSO_vertical := 500;
END_DATA_BLOCK

DATA_BLOCK "gtyp_SetupAxis"   // DB4
TITLE = Global DB Setup Axis
{ S7_Optimized_Access := 'TRUE' }
AUTHOR : A.Schaefer
VERSION : 0.0
BEGIN
END_DATA_BLOCK

DATA_BLOCK "gtyp_MPO"   // DB11
TITLE = Global DB MPO
{ S7_Optimized_Access := 'TRUE' }
AUTHOR : A.Schaefer
VERSION : 0.0
BEGIN
END_DATA_BLOCK

DATA_BLOCK "gtyp_SSC"   // DB13
TITLE = Global DB SSC
{ S7_Optimized_Access := 'TRUE' }
AUTHOR : A.Schaefer
VERSION : 0.0
BEGIN
   Horizontal_Axis.Config.di_Pos_Soft_Switch := 5450;
   Vertical_Axis.Config.di_Pos_Soft_Switch := 3000;
   di_Pos_Centre_Horizontal := 3000;
   di_Pos_Centre_Vertical := 1400;
   Vertical_Axis.Config.di_Pos_Window := 25;
   Horizontal_Axis.Config.di_Pos_Window := 25;
   di_Pos_HBW_Horizontal := 5400;
   di_Pos_HBW_Vertical := 950;
   Horizontal_Axis.i_PWM := 1000;
   Vertical_Axis.i_PWM := 1000;
   w_Threshold_White_Red := 16#25DA;
   w_Threshold_Red_Blue := 16#3C57;
END_DATA_BLOCK

DATA_BLOCK "gtyp_HBW"   // DB17
TITLE = Global DB HBW
{ S7_Optimized_Access := 'TRUE' }
AUTHOR : A.Schaefer
VERSION : 0.0
BEGIN
   Horizontal_Axis.Config.di_Pos_Soft_Switch := 7900;
   Vertical_Axis.Config.di_Pos_Soft_Switch := 3350;
   di_PosBelt_Vertical := 2800;
   di_PosBelt_Horizontal := 18;
   di_Offset_Pos_Belt_Vertical := 370;
   Rack_Pos[1,1].di_PosRack_Horizontal := 2870;
   Rack_Pos[1,1].di_PosRack_Vertical := 400;
   Rack_Pos[1,2].di_PosRack_Horizontal := 5200;
   Rack_Pos[1,2].di_PosRack_Vertical := 400;
   Rack_Pos[1,3].di_PosRack_Horizontal := 7550;
   Rack_Pos[1,3].di_PosRack_Vertical := 400;
   Rack_Pos[2,1].di_PosRack_Horizontal := 2870;
   Rack_Pos[2,2].di_PosRack_Horizontal := 5200;
   Rack_Pos[2,3].di_PosRack_Horizontal := 7550;
   Rack_Pos[2,1].di_PosRack_Vertical := 1750;
   Rack_Pos[2,2].di_PosRack_Vertical := 1750;
   Rack_Pos[2,3].di_PosRack_Vertical := 1750;
   Rack_Pos[3,1].di_PosRack_Horizontal := 2870;
   Rack_Pos[3,1].di_PosRack_Vertical := 3150;
   Rack_Pos[3,2].di_PosRack_Horizontal := 5200;
   Rack_Pos[3,2].di_PosRack_Vertical := 3150;
   Rack_Pos[3,3].di_PosRack_Horizontal := 7550;
   Rack_Pos[3,3].di_PosRack_Vertical := 3150;
   Horizontal_Axis.Config.di_Pos_Window := 15;
   Vertical_Axis.Config.di_Pos_Window := 15;
   Horizontal_Axis.i_PWM := 700;
   Vertical_Axis.i_PWM := 600;
   Rack_Workpiece[1,1].s_id := '0';
   Rack_Workpiece[1,2].s_id := '0';
   Rack_Workpiece[1,3].s_id := '0';
   Rack_Workpiece[2,1].s_id := '0';
   Rack_Workpiece[2,2].s_id := '0';
   Rack_Workpiece[2,3].s_id := '0';
   Rack_Workpiece[3,1].s_id := '0';
   Rack_Workpiece[3,2].s_id := '0';
   Rack_Workpiece[3,3].s_id := '0';
   di_PosRack_A1_Horizontal := 2870;
   di_PosRack_A1_Vertical := 400;
   di_PosRack_B2_Horizontal := 5200;
   di_PosRack_B2_Vertical := 1750;
   di_PosRack_C3_Horizontal := 7560;
   di_PosRack_C3_Vertical := 3250;
   di_Offset_Pos_Rack_Vertical := 370;
   i_PWM_Cantilever := 1000;
END_DATA_BLOCK

DATA_BLOCK "gtyp_Setup"   // DB23
TITLE = Global DB Setup
{ S7_Optimized_Access := 'TRUE' }
AUTHOR : A.Schaefer
VERSION : 0.0
BEGIN
END_DATA_BLOCK

DATA_BLOCK "gtyp_SLD"   // DB24
TITLE = Global DB SLD
{ S7_Optimized_Access := 'TRUE' }
AUTHOR : A.Schaefer
VERSION : 0.0
BEGIN
   i_CounterValue_White := 5;
   i_CounterValue_Blue := 26;
   i_CounterValue_Red := 16;
   w_Threshold_White_Red := 16#2698;
   w_Threshold_Red_Blue := 16#3D41;
END_DATA_BLOCK

DATA_BLOCK "gtyp_Interface_TXT_Controler"   // DB40
{ S7_Optimized_Access := 'TRUE' }
VERSION : 0.1
BEGIN
END_DATA_BLOCK

DATA_BLOCK "RT_INFO_scl_OB30"   // DB325
{ S7_Optimized_Access := 'TRUE' }
VERSION : 0.1
   VAR
      mode : UInt := 1;   // Mode 1 = Runtime of a specific OB; 2 = Maximum runtime of a specific OB; 3 = Minimum runtime of a specific OB; 10 = Mean value of the percentage of total runtime used by higher-priority OBs; ...
      obNbr : OB_Any := 1;   // OB to read
      infoData : LTime;   // mode 1 --> Runtime in LTIME
      returnValue : Int;   // Error information of instruction
   END_VAR
BEGIN
END_DATA_BLOCK

DATA_BLOCK "RT_INFO_scl_OB1"   // DB326
{ S7_Optimized_Access := 'TRUE' }
VERSION : 0.1
   VAR
      mode : UInt := 1;   // Mode 1 = Runtime of a specific OB; 2 = Maximum runtime of a specific OB; 3 = Minimum runtime of a specific OB; 10 = Mean value of the percentage of total runtime used by higher-priority OBs; ...
      obNbr : OB_Any := 1;   // OB to read
      infoData : LTime;   // mode 1 --> Runtime in LTIME
      returnValue : Int;   // Error information of instruction
   END_VAR
BEGIN
END_DATA_BLOCK

// folder: (top level)

ORGANIZATION_BLOCK "Main"   // OB1, SCL, ProgramCycle
TITLE = "Main Program Sweep (Cycle)"
{ S7_Optimized_Access := 'TRUE' }
AUTHOR : A.Schaefer
VERSION : 0.0
   VAR_INPUT
      Initial_Call : Bool;   // Initial call of this OB
      Remanence : Bool;   // =True, if remanent data are available
   END_VAR
BEGIN
   // current cycle Time OB30
   "RT_INFO_scl_OB30".mode := 1;
   "RT_INFO_scl_OB30".obNbr := 30;
   "RT_INFO_scl_OB30".returnValue := RT_INFO(MODE := "RT_INFO_scl_OB30".mode,
                                             OB := "RT_INFO_scl_OB30".obNbr,
                                             INFO := "RT_INFO_scl_OB30".infoData);

   // current cycle Time OB1
   "RT_INFO_scl_OB1".mode := 1;
   "RT_INFO_scl_OB1".obNbr := 1;
   "RT_INFO_scl_OB1".returnValue := RT_INFO(MODE := "RT_INFO_scl_OB1".mode,
                                            OB := "RT_INFO_scl_OB1".obNbr,
                                            INFO := "RT_INFO_scl_OB1".infoData);

   // sources SSC
   "PRG_SSC_Ablauf_DB"();
   "PRG_SSC_Set_Positioning_DB"();
   "PRG_SSC_Calibration_Color_DB"();
   "PRG_SSC_Axis_Vertical_DB"();
   "PRG_SSC_Axis_Horizontal_DB"();
   "PRG_SSC_Light_DB"();

   // sources VGR
   "PRG_VGR_Ablauf_DB"();
   "PRG_VGR_Set_Positioning_DB"();
   "PRG_VGR_Axis_horizontal_DB"();
   "PRG_VGR_Axis_vertical_DB"();
   "PRG_VGR_Axis_rotate_DB"();
   "PRG_NFC_DB"();

   // sources HBW
   "PRG_HBW_Ablauf_DB"();
   "PRG_HBW_Set_Positioning_DB"();
   "PRG_HBW_Axis_Vertical_DB"();
   "PRG_HBW_Axis_Horizontal_DB"();

   // sources MPO
   "PRG_MPO_Ablauf_DB"();

   // sources SLD
   "PRG_SLD_Ablauf_DB"();
   "PRG_SLD_Calibration_Color_DB"();
   "PRG_SLD_Set_Counter_Values_DB"();

   // sources input/output
   "PRG_DSI_Status_DB"();
   "PRG_DSO_Status_DB"();

   // sources dashboard
   "PRG_Order_DB"();
   "PRG_Acknowledge_DB"();
END_ORGANIZATION_BLOCK

ORGANIZATION_BLOCK "Cyclic interrupt"   // OB30, SCL, CyclicInterrupt
TITLE = Cyclic interrupt
{ S7_Optimized_Access := 'TRUE' }
AUTHOR : A.Schaefer
VERSION : 0.0
   VAR_INPUT
      Initial_Call : Bool;   // Initial call of this OB
      Event_Count : Int;   // Events discarded
   END_VAR
   VAR_TEMP
      li_Return_LDT : Int;
   END_VAR
BEGIN

   "PRG_SSC_Axis_Horizontal_Act_Pos_DB"();
   "PRG_SSC_Axis_Vertical_Act_Pos_DB"();

   "PRG_HBW_Axis_Horizontal_Act_Pos_DB"();
   "PRG_HBW_Axis_Vertical_Act_Pos_DB"();

   "PRG_VGR_Axis_horizontal_Act_Pos_DB"();
   "PRG_VGR_Axis_vertical_Act_Pos_DB"();
   "PRG_VGR_Axis_rotate_Act_Pos_DB"();
END_ORGANIZATION_BLOCK

// folder: 1. FB / FC

FUNCTION_BLOCK "FB_Blinker"   // FB2, SCL
TITLE = Functionblock Blinker
{ S7_Optimized_Access := 'TRUE' }
AUTHOR : A.Schaefer
VERSION : 0.0
   VAR_INPUT
      int_periodendauer : Time;
   END_VAR
   VAR_OUTPUT
      outx_blinker : Bool;
   END_VAR
   VAR
      lfb_ton : TON_TIME;
      lx_esv_timer : Bool;
      lx_blinker : Bool;
   END_VAR
BEGIN
   #lfb_ton(IN := NOT #lx_esv_timer,
           PT := #int_periodendauer / 2,
           Q => #lx_esv_timer);

   IF #lx_esv_timer THEN
       #lx_blinker := NOT #lx_blinker;
   END_IF;

   #outx_blinker := #lx_blinker;
END_FUNCTION_BLOCK

FUNCTION_BLOCK "FB_INC_DEC"   // FB9, SCL
TITLE = Funktionblock Increment decodition
{ S7_Optimized_Access := 'TRUE' }
AUTHOR : A.Schaefer
VERSION : 0.0
   VAR_INPUT
      inx_CHa : Bool := false;
      inx_CHb : Bool := false;
      inx_RST : Bool := False;
      ini_Ref_Wert : Int := 0;
   END_VAR
   VAR_OUTPUT
      outx_dir : Bool := false;
      outi_cnt : Int := 0;
   END_VAR
   VAR
      lx_edgea : Bool := False;
      lx_clka : Bool;
      lx_clkb : Bool;
      lx_edgeb : Bool;
      lx_axb : Bool;
      lx_dir : Bool;
      li_cnt : Int;
   END_VAR
BEGIN

   #lx_axb := #inx_CHa XOR #inx_CHb;

   (* create pulses for channel a *)
   #lx_clka := #inx_CHa XOR #lx_edgea;
   #lx_edgea := #inx_CHa;

   #lx_clkb := #inx_CHb XOR #lx_edgeb;
   #lx_edgeb := #inx_CHb;

   (* create pulses for both channels *)
   #lx_clka := #lx_clka OR #lx_clkb;

   (* set the direction output *)
   IF #lx_axb AND #lx_clka THEN
       #lx_dir := TRUE;
   END_IF;
   IF #lx_axb AND #lx_clkb THEN
       #lx_dir := FALSE;
   END_IF;

   (* increment or decrement the counter *)
   IF #lx_clka AND #lx_dir THEN
       #li_cnt := #li_cnt + 1;
   END_IF;
   IF #lx_clka AND NOT #lx_dir THEN
       #li_cnt := #li_cnt - 1;
   END_IF;

   (* reset the counter if rst active *)
   IF #inx_RST THEN
       #li_cnt := #ini_Ref_Wert;
   END_IF;

   #outx_dir := #lx_dir;
   #outi_cnt := #li_cnt;
END_FUNCTION_BLOCK

FUNCTION_BLOCK "FB_Axis"   // FB22, SCL
TITLE = Functionblock Axis
{ S7_Optimized_Access := 'TRUE' }
AUTHOR : A.Schaefer
VERSION : 0.0
   VAR_INPUT
      ini_Axis : Int;
      indi_Increment : DInt;
      inx_Ref_Switch : Bool;
      inx_Start_Positioning : Bool;
      inx_Referencing : Bool;
      ini_PWM : Int;
      indi_Target_Position : DInt;
   END_VAR
   VAR_OUTPUT
      outx_Referenced : Bool;
      outx_Position_Reached : Bool;
      outx_Motor_Pos : Bool;
      outx_Motor_Neg : Bool;
      outi_Motor_PWM : Int;
      outdi_Actual_Position : DInt;
   END_VAR
   VAR_IN_OUT
      inouttyp_Config : "typ_Axis_Data";
      inouttyp_Setup : "typ_SetupAxis";
   END_VAR
   VAR
      li_StepCaseSetup : Int;
      li_StepCase : Int;
      lx_Init : Bool;
      lx_Motor_Neg : Bool;
      lx_Motor_Pos : Bool;
      lx_Start_TON_Wait : Bool;
      li_PWM : Int;
      ldi_ValueStep : DInt;
      ldi_Actual_Position : DInt;
      ldi_Actual_Position_Old : DInt;
      lfb_R_Trig_Setup : R_TRIG;
      lfb_R_Trig_Referencing : R_TRIG;
      lfb_TON_Wait : TON_TIME;
   END_VAR
BEGIN
   IF #lx_Init THEN

       // rising edge set up axis
       #lfb_R_Trig_Setup(CLK := #inouttyp_Setup.x_Setup_Activ);

       //Reload when switching to set up
       IF #lfb_R_Trig_Setup.Q THEN
           #inouttyp_Setup.di_LoopValue               := #inouttyp_Config.di_Loop_Value;
           #inouttyp_Setup.di_Ref_Pos                 := 
           #inouttyp_Setup.di_Actual_Ref_Pos          := #inouttyp_Config.di_Ref_Pos;
           #inouttyp_Setup.di_Soft_End_Pos_Neg        := 
           #inouttyp_Setup.di_Actual_Soft_End_Pos_Neg := #inouttyp_Config.di_Neg_Soft_Switch;
           #inouttyp_Setup.di_Soft_End_Pos_Pos        :=
           #inouttyp_Setup.di_Actual_Soft_End_Pos_Pos := #inouttyp_Config.di_Pos_Soft_Switch;
           #inouttyp_Setup.i_PWM                      := #ini_PWM;
           #inouttyp_Setup.x_Approach_Ref_Pos         := FALSE;
           #inouttyp_Setup.x_Approach_Target_Pos      := FALSE;
           #inouttyp_Setup.x_Axis_Neg                 := FALSE;
           #inouttyp_Setup.x_Axis_Pos                 := FALSE;
           #inouttyp_Setup.x_Set_Ref_Pos              := FALSE;
           #inouttyp_Setup.x_Set_Soft_End_Pos         := FALSE;
       END_IF;

       #ldi_Actual_Position := #indi_Increment;

       //rising edge referencing
       #lfb_R_Trig_Referencing(CLK := #inx_Referencing);

       //waiting period
       #lfb_TON_Wait(IN := #lx_Start_TON_Wait,
                     PT := T#200ms);

       (**********************************)
       (******   set up step chain   *****)
       (**********************************)
       IF #inouttyp_Setup.i_AxisSelection = #ini_Axis AND #inouttyp_Setup.x_Setup_Activ THEN
           IF #inouttyp_Setup.x_Approach_Ref_Pos THEN
               #inouttyp_Setup.i_Function := 10;
           END_IF;

           CASE #inouttyp_Setup.i_Function OF

               0:  // automatic
                   #ldi_Actual_Position_Old := 0;
                   #inouttyp_Setup.x_Approach_Ref_Pos := FALSE;
                   #lx_Start_TON_Wait := FALSE;

               10: // homing
                   IF #inouttyp_Setup.x_Approach_Ref_Pos THEN
                       IF NOT #inx_Ref_Switch THEN
                           #lx_Motor_Neg := TRUE;
                           #lx_Motor_Pos := FALSE;
                           #outx_Referenced := FALSE;
                       END_IF;

                       IF #inx_Ref_Switch THEN
                           #lx_Motor_Neg := TRUE;
                           #lx_Motor_Pos := TRUE;

                           IF #ldi_Actual_Position = #inouttyp_Config.di_Ref_Pos THEN
                               #inouttyp_Setup.x_Approach_Ref_Pos := FALSE;
                               #lx_Motor_Neg       := FALSE;
                               #lx_Motor_Pos       := FALSE;
                               #outx_Referenced    := TRUE;
                           END_IF;
                       END_IF;
                   END_IF;

               20:  // tap
                   #lx_Motor_Neg := #inouttyp_Setup.x_Axis_Neg AND NOT #inx_Ref_Switch AND NOT (#ldi_Actual_Position <= #inouttyp_Setup.di_Soft_End_Pos_Neg);
                   #lx_Motor_Pos := #inouttyp_Setup.x_Axis_Pos AND NOT #lx_Motor_Neg AND NOT (#ldi_Actual_Position >= #inouttyp_Setup.di_Soft_End_Pos_Pos);

               30:  // tap with increment
                   #ldi_Actual_Position_Old := #ldi_Actual_Position;

                   // positiv
                   IF #inouttyp_Setup.x_Axis_Pos AND NOT ((#ldi_Actual_Position + #inouttyp_Setup.w_Increment + #inouttyp_Setup.di_LoopValue) >= #inouttyp_Setup.di_Soft_End_Pos_Pos) THEN
                       #lx_Motor_Neg := FALSE;
                       #lx_Motor_Pos := TRUE;
                       #ldi_ValueStep := #ldi_Actual_Position_Old + #inouttyp_Setup.w_Increment;

                       // without loop
                       IF (#inouttyp_Setup.di_LoopValue = 0) THEN
                           #inouttyp_Setup.i_Function := 36;
                       ELSE
                           #inouttyp_Setup.i_Function := 31;
                       END_IF;
                   // negativ
                   ELSIF #inouttyp_Setup.x_Axis_Neg AND NOT ((#ldi_Actual_Position - #inouttyp_Setup.w_Increment) <= #inouttyp_Config.di_Neg_Soft_Switch) THEN
                       #lx_Motor_Neg := TRUE;
                       #lx_Motor_Pos := FALSE;
                       #ldi_ValueStep := #ldi_Actual_Position_Old - #inouttyp_Setup.w_Increment;
                       #inouttyp_Setup.i_Function := 34;
                   END_IF;

               31: // with loop
                   IF ((#ldi_Actual_Position >= (#ldi_ValueStep + #inouttyp_Setup.di_LoopValue - #inouttyp_Config.di_Pos_Window)) = 0) THEN
                       #lx_Motor_Neg := TRUE;
                       #lx_Motor_Pos := TRUE;
                       #inouttyp_Setup.i_Function := 32;
                   END_IF;

               32: // wait sequence
                   #lx_Start_TON_Wait := TRUE;

                   IF #lfb_TON_Wait.Q THEN
                       #lx_Motor_Neg               := FALSE;
                       #lx_Motor_Pos               := FALSE;
                       #lx_Start_TON_Wait          := FALSE;
                       #inouttyp_Setup.i_Function  := 33;
                   END_IF;

               33: // change direction
                   #lx_Motor_Neg := TRUE;
                   #lx_Motor_Pos := FALSE;
                   #inouttyp_Setup.i_Function := 34;

               34: // position reached negativ
                   IF (#ldi_Actual_Position <= (#ldi_ValueStep + #inouttyp_Config.di_Pos_Window))
                       AND (#ldi_Actual_Position >= (#ldi_ValueStep - #inouttyp_Config.di_Pos_Window)) THEN
                       #lx_Motor_Neg := TRUE;
                       #lx_Motor_Pos := TRUE;
                       #inouttyp_Setup.i_Function := 35;
                   END_IF;

               35: // wait sequence
                   #lx_Start_TON_Wait := TRUE;

                   IF #lfb_TON_Wait.Q THEN
                       #lx_Motor_Neg := FALSE;
                       #lx_Motor_Pos := FALSE;
                       #lx_Start_TON_Wait := FALSE;
                       #inouttyp_Setup.x_Axis_Neg := FALSE;
                       #inouttyp_Setup.x_Axis_Pos := FALSE;
                       #inouttyp_Setup.i_Function := 30;
                   END_IF;


               36: // position reached positiv
                   IF (#ldi_Actual_Position <= (#ldi_ValueStep + #inouttyp_Config.di_Pos_Window))
                       AND (#ldi_Actual_Position >= (#ldi_ValueStep - #inouttyp_Config.di_Pos_Window)) THEN
                       #lx_Motor_Neg := TRUE;
                       #lx_Motor_Pos := TRUE;
                       #inouttyp_Setup.i_Function := 37;
                   END_IF;

               37: // wait sequence
                   #lx_Start_TON_Wait := TRUE;

                   IF #lfb_TON_Wait.Q THEN
                       #lx_Motor_Neg := FALSE;
                       #lx_Motor_Pos := FALSE;
                       #lx_Start_TON_Wait := FALSE;
                       #inouttyp_Setup.x_Axis_Neg := FALSE;
                       #inouttyp_Setup.x_Axis_Pos := FALSE;
                       #inouttyp_Setup.i_Function := 30;
                   END_IF;

               40: // approach position
                   IF #inouttyp_Setup.x_Approach_Target_Pos THEN
                       // positiv
                       IF (#inouttyp_Setup.di_Target_Position > #ldi_Actual_Position) AND NOT ((#inouttyp_Setup.di_Target_Position + #inouttyp_Setup.di_LoopValue) >= #inouttyp_Setup.di_Soft_End_Pos_Pos)  THEN
                           #lx_Motor_Neg := FALSE;
                           #lx_Motor_Pos := TRUE;
                           // without loop
                           IF (#inouttyp_Setup.di_LoopValue = 0) THEN
                               #inouttyp_Setup.i_Function := 46;
                           ELSE
                               #inouttyp_Setup.i_Function := 41;
                           END_IF;
                       // negativ
                       ELSIF ((#inouttyp_Setup.di_Target_Position < #ldi_Actual_Position) AND NOT (#inouttyp_Setup.di_Target_Position <= #inouttyp_Config.di_Neg_Soft_Switch))  THEN
                           #lx_Motor_Neg := TRUE;
                           #lx_Motor_Pos := FALSE;
                           #inouttyp_Setup.i_Function := 44;
                       ELSIF (#inouttyp_Setup.di_Target_Position = #ldi_Actual_Position) THEN
                           #inouttyp_Setup.i_Function := 46;
                       END_IF;

                   END_IF;

               41: // with loop
                   IF (#ldi_Actual_Position >= (#inouttyp_Setup.di_Target_Position + #inouttyp_Setup.di_LoopValue - #inouttyp_Config.di_Pos_Window)) THEN
                       #lx_Motor_Neg := TRUE;
                       #lx_Motor_Pos := TRUE;
                       #inouttyp_Setup.i_Function := 42;
                   END_IF;

               42: // wait sequence
                   #lx_Start_TON_Wait := TRUE;

                   IF #lfb_TON_Wait.Q THEN
                       #lx_Motor_Neg := FALSE;
                       #lx_Motor_Pos := FALSE;
                       #lx_Start_TON_Wait := FALSE;
                       #inouttyp_Setup.i_Function := 43;
                   END_IF;

               43: // change direction
                   #lx_Motor_Neg   := TRUE;
                   #lx_Motor_Pos   := FALSE;
                   #inouttyp_Setup.i_Function     := 44;

               44: // position reached negativ
                   IF (#ldi_Actual_Position <= (#inouttyp_Setup.di_Target_Position + #inouttyp_Config.di_Pos_Window))
                       AND (#ldi_Actual_Position >= (#inouttyp_Setup.di_Target_Position - #inouttyp_Config.di_Pos_Window)) THEN
                       #lx_Motor_Neg := TRUE;
                       #lx_Motor_Pos := TRUE;
                       #inouttyp_Setup.i_Function := 45;
                   END_IF;

               45: // wait sequence
                   #lx_Start_TON_Wait := TRUE;

                   IF #lfb_TON_Wait.Q THEN
                       #lx_Motor_Neg := FALSE;
                       #lx_Motor_Pos := FALSE;
                       #lx_Start_TON_Wait := FALSE;
                       #inouttyp_Setup.x_Axis_Neg := FALSE;
                       #inouttyp_Setup.x_Axis_Pos := FALSE;
                       #inouttyp_Setup.i_Function := 40;
                   END_IF;

               46: //  position reached positiv
                   IF (#ldi_Actual_Position <= (#inouttyp_Setup.di_Target_Position + #inouttyp_Config.di_Pos_Window))
                       AND (#ldi_Actual_Position >= (#inouttyp_Setup.di_Target_Position - #inouttyp_Config.di_Pos_Window)) THEN
                       #lx_Motor_Neg := TRUE;
                       #lx_Motor_Pos := TRUE;
                       #inouttyp_Setup.i_Function := 47;
                   END_IF;

               47:  // wait sequence
                   #lx_Start_TON_Wait := TRUE;

                   IF #lfb_TON_Wait.Q THEN
                       #lx_Motor_Neg := FALSE;
                       #lx_Motor_Pos := FALSE;
                       #lx_Start_TON_Wait := FALSE;
                       #inouttyp_Setup.x_Approach_Target_Pos := FALSE;
                       #inouttyp_Setup.i_Function := 40;
                   END_IF;
               ELSE  // Statement section ELSE
                   ;
           END_CASE;

           // set reference point
           IF #inouttyp_Setup.x_Set_Ref_Pos THEN
               #inouttyp_Setup.di_Actual_Ref_Pos   :=
               #inouttyp_Config.di_Ref_Pos         := #inouttyp_Setup.di_Ref_Pos;
               #inouttyp_Setup.x_Set_Ref_Pos       := FALSE;
           END_IF;

           // set software end position
           IF #inouttyp_Setup.x_Set_Soft_End_Pos THEN
               #inouttyp_Setup.di_Actual_Soft_End_Pos_Neg  :=
               #inouttyp_Config.di_Neg_Soft_Switch         := #inouttyp_Setup.di_Soft_End_Pos_Neg;
               #inouttyp_Setup.di_Actual_Soft_End_Pos_Pos  :=
               #inouttyp_Config.di_Pos_Soft_Switch         := #inouttyp_Setup.di_Soft_End_Pos_Pos;
               #inouttyp_Setup.x_Set_Soft_End_Pos := FALSE;
           END_IF;

           // reload PWM
           #li_PWM := #inouttyp_Setup.i_PWM;

           // reload actual position
           #inouttyp_Setup.di_ActualPosition           := #ldi_Actual_Position;

       (************************************)
       (******   position step chain   *****)
       (************************************)
       ELSIF NOT #inouttyp_Setup.x_Setup_Activ THEN

           // rising edge set up axis
           IF #lfb_R_Trig_Referencing.Q THEN
               #li_StepCase := 0;
           END_IF;

           CASE #li_StepCase OF

               0:  // init
                   #lx_Start_TON_Wait := FALSE;

                   IF #inx_Referencing THEN
                       #li_StepCase            := 10;
                       #outx_Position_Reached  := FALSE;
                       #outx_Referenced        := FALSE;
                   ELSIF #inx_Start_Positioning THEN
                       #li_StepCase            := 20;
                       #outx_Position_Reached  := FALSE;
                   END_IF;

               10: // homing
                   IF NOT #inx_Ref_Switch THEN
                       #lx_Motor_Neg := TRUE;
                       #lx_Motor_Pos := FALSE;
                   END_IF;

                   IF #inx_Ref_Switch THEN
                       #lx_Motor_Neg := TRUE;
                       #lx_Motor_Pos := TRUE;

                       IF #inx_Ref_Switch THEN
                           IF #ldi_Actual_Position = #inouttyp_Config.di_Ref_Pos THEN
                               #lx_Motor_Neg := FALSE;
                               #lx_Motor_Pos := FALSE;
                               #outx_Referenced := TRUE;
                               #li_StepCase := 11;
                           END_IF;
                       END_IF;
                   END_IF;

               11: // wait not referencing
                   IF NOT #inx_Referencing THEN
                       #li_StepCase := 0;
                   END_IF;

               20: // approach position
                   // positiv
                   IF (#indi_Target_Position > #ldi_Actual_Position) AND NOT ((#indi_Target_Position + #inouttyp_Config.di_Loop_Value) >= #inouttyp_Config.di_Pos_Soft_Switch) THEN
                       #lx_Motor_Neg := FALSE;
                       #lx_Motor_Pos := TRUE;
                       //without loop
                       IF (#inouttyp_Config.di_Loop_Value = 0) THEN
                           #li_StepCase := 26;
                       ELSE
                           #li_StepCase := 21;
                       END_IF;
                   // negativ
                   ELSIF ((#indi_Target_Position < #ldi_Actual_Position) AND NOT (#indi_Target_Position <= #inouttyp_Config.di_Neg_Soft_Switch)) THEN
                       #lx_Motor_Neg := TRUE;
                       #lx_Motor_Pos := FALSE;
                       #li_StepCase := 24;
                   ELSIF (#indi_Target_Position = #ldi_Actual_Position) THEN
                       #li_StepCase := 26;
                   END_IF;

               21: // with loop
                   IF (#ldi_Actual_Position >= (#indi_Target_Position + #inouttyp_Config.di_Loop_Value - #inouttyp_Config.di_Pos_Window)) THEN
                       #lx_Motor_Neg := TRUE;
                       #lx_Motor_Pos := TRUE;
                       #li_StepCase := 22;
                   END_IF;

               22: // wait sequence
                   #lx_Start_TON_Wait := TRUE;

                   IF #lfb_TON_Wait.Q THEN
                       #lx_Motor_Neg := FALSE;
                       #lx_Motor_Pos := FALSE;
                       #lx_Start_TON_Wait := FALSE;
                       #inouttyp_Setup.i_Function := 23;
                   END_IF;

               23: // change direction
                   #lx_Motor_Neg := TRUE;
                   #lx_Motor_Pos := FALSE;
                   #li_StepCase := 24;

               24: // position reached negativ
                   IF (#ldi_Actual_Position <= (#indi_Target_Position + #inouttyp_Config.di_Pos_Window))
                       AND (#ldi_Actual_Position >= (#indi_Target_Position - #inouttyp_Config.di_Pos_Window)) THEN
                       #lx_Motor_Neg := TRUE;
                       #lx_Motor_Pos := TRUE;
                       #li_StepCase := 25;
                   END_IF;

               25: // wait sequence
                   #lx_Start_TON_Wait := TRUE;

                   IF #lfb_TON_Wait.Q THEN
                       #lx_Motor_Neg := FALSE;
                       #lx_Motor_Pos := FALSE;
                       #lx_Start_TON_Wait := FALSE;
                       #outx_Position_Reached := TRUE;
                       #li_StepCase := 28;
                   END_IF;

               26: // position reached positiv
                   IF (#ldi_Actual_Position <= (#indi_Target_Position + #inouttyp_Config.di_Pos_Window))
                       AND (#ldi_Actual_Position >= (#indi_Target_Position - #inouttyp_Config.di_Pos_Window)) THEN
                       #lx_Motor_Neg := TRUE;
                       #lx_Motor_Pos := TRUE;
                       #li_StepCase := 27;
                   END_IF;

               27: // wait sequence
                   #lx_Start_TON_Wait := TRUE;

                   IF #lfb_TON_Wait.Q THEN
                       #lx_Motor_Neg := FALSE;
                       #lx_Motor_Pos := FALSE;
                       #lx_Start_TON_Wait := FALSE;
                       #outx_Position_Reached := TRUE;
                       #li_StepCase := 28;
                   END_IF;

               28: // wait not start positioning
                   IF NOT #inx_Start_Positioning THEN
                       #li_StepCase := 0;
                   END_IF;
               // statement section ELSE    
               ELSE  
                   ;
           END_CASE;

           // reload PWM
           #li_PWM := #ini_PWM;
       END_IF;

       // reload outputs
       #outx_Motor_Neg         := #lx_Motor_Neg;
       #outx_Motor_Pos         := #lx_Motor_Pos;
       #outi_Motor_PWM         := #li_PWM;
       #outdi_Actual_Position  := #ldi_Actual_Position;

   ELSE
       #lx_Init := TRUE;
   END_IF;
END_FUNCTION_BLOCK

FUNCTION "FC_Scale_linear" : Real   // FC1, SCL
TITLE = Function scale linear
{ S7_Optimized_Access := 'TRUE' }
AUTHOR : A.Schaefer
VERSION : 0.0
   VAR_INPUT
      inr_Y1 : Real;   // Skalierungs-Anfangswert für Y (OUTPUT) / Initial scaling value for Y (INPUT)
      inr_Y2 : Real;   // Skalierungs-Endwert für Y (OUTPUT) / Scaling end value for Y (INPUT)
      inr_X1 : Real;   // Skalierungs-Anfangswert für X (INPUT) / Initial scaling value for X (INPUT)
      inr_X2 : Real;   // Skalierungs-Endwert für X (INPUT) / Scaling end value for X (INPUT)
      inr_X : Real;   // Zu Skalierender Wert / Value to be scaled
   END_VAR
   VAR_TEMP
      lr_y_delta : Real;   // Temp delta y
      lr_x_delta : Real;   // Temp delta x
      lr_m : Real;   // Temp gradient m
   END_VAR
   // Ret_Val : Return result
BEGIN
   (********************************************************)
   (* FC for linear scaling. Line function  y=m*(x-x1)+y1  *)
   (********************************************************)

   #lr_y_delta := (#inr_Y2 - #inr_Y1);
   #lr_x_delta := (#inr_X2 - #inr_X1);

   IF #lr_y_delta <> 0 AND #lr_x_delta <> 0 THEN
       #lr_m := (#lr_y_delta / #lr_x_delta);
       #FC_Scale_linear := (#lr_m * (#inr_X - #inr_X1)) + #inr_Y1;
   ELSE
       #FC_Scale_linear := 0;
   END_IF;
END_FUNCTION

// folder: 2. Cloud

FUNCTION_BLOCK "PRG_NFC"   // FB8, SCL
TITLE = Program NFC
{ S7_Optimized_Access := 'TRUE' }
AUTHOR : A.Schaefer
VERSION : 0.0
   VAR
      lx_Init : Bool;
      lx_Start : Bool;
      lx_Time_Wait : Bool;
      lx_Time_Error : Bool;
      li_StepCase : Int;
      ldt_MQTT : Date_And_Time;
      ldt_Delete_old : LDT;
      ldt_Read_old : LDT;
      li_Return_LDT : Int;
      lfb_TON_Error : TON_TIME;
      lfb_TON_Wait : TON_TIME;
   END_VAR
BEGIN
   IF #lx_Init THEN

       // runtime monitoring error
       #lfb_TON_Error(IN:= #lx_Time_Error,
                      PT:= T#30s);

       // runtime monitoring read uid
       #lfb_TON_Wait(IN := #lx_Time_Wait,
                     PT := T#5s);

        // step chain NFC
       CASE #li_StepCase OF

           0:  // init
               #lx_Time_Wait                := FALSE;
               "gtyp_VGR"."x_NFC_Completed" := FALSE;

               // delete and write first state to chip
               IF "gtyp_VGR".x_NFC_Start_First AND NOT "gtyp_VGR".x_Workpiece_NiO THEN
                   "gtyp_Interface_TXT_Controler".Subscribe.State_NFC_Device.Workpiece.s_state := '';
                   "gtyp_Interface_TXT_Controler".Subscribe.State_NFC_Device.Workpiece.s_type := '';

                   "gtyp_Interface_TXT_Controler".Publish.ActionButtonNFCModule.s_cmd := '';
                   #li_StepCase := 10;
                   // write color or processed finished to chip
               ELSIF "gtyp_VGR".x_NFC_Start AND NOT "gtyp_VGR".x_Workpiece_NiO THEN
                   "gtyp_Interface_TXT_Controler".Publish.ActionButtonNFCModule.s_cmd := '';
                   #li_StepCase := 40;
                   // read chip for delete HBW
               ELSIF "QX_SSC_LED_Green_Q5" AND NOT "gtyp_VGR".x_Workpiece_NiO THEN
                   #ldt_Read_old := "gtyp_Interface_Dashboard".Publish.ActionButtonNFCModule.ldt_ts;
                   "gtyp_VGR".x_NFC_Start_First := FALSE;
                   "gtyp_VGR".x_NFC_Start := FALSE;
                   "gtyp_Interface_TXT_Controler".Publish.ActionButtonNFCModule.s_cmd := '';
                   #li_StepCase := 60;
               END_IF;

           10: // delete

               "gtyp_Interface_TXT_Controler".Publish.ActionButtonNFCModule.s_cmd := 'delete';
               #li_Return_LDT := RD_SYS_T(#ldt_MQTT);
               "gtyp_Interface_TXT_Controler".Publish.ActionButtonNFCModule.ldt_ts := DT_TO_LDT(#ldt_MQTT);

               #li_StepCase := 20;

           20: // wait to answer from dashboard
               #lx_Time_Error := TRUE;
               IF ("gtyp_Interface_TXT_Controler".Subscribe.State_NFC_Device.ldt_ts > "gtyp_Interface_TXT_Controler".Publish.ActionButtonNFCModule.ldt_ts)
                   AND ("gtyp_Interface_TXT_Controler".Subscribe.State_NFC_Device.Workpiece.s_type = 'NONE')
                   AND ("gtyp_Interface_TXT_Controler".Subscribe.State_NFC_Device.Workpiece.s_state <> '')
                   AND ("gtyp_Interface_TXT_Controler".Subscribe.State_NFC_Device.Workpiece.s_id <> '') THEN
                   "gtyp_VGR".Workpiece.s_id := "gtyp_Interface_TXT_Controler".Subscribe.State_NFC_Device.Workpiece.s_id;
                   #lx_Time_Error := FALSE;
                   #li_StepCase := 30;
               END_IF;
               // runtime error
               IF #lfb_TON_Error.Q THEN
                   #lx_Time_Error := FALSE;
                   "gtyp_VGR".x_Workpiece_NiO := TRUE;
                   #li_StepCase := 0;
               END_IF;


           30: // wait of answer 
               IF "gtyp_Interface_TXT_Controler".Subscribe.State_NFC_Device.Workpiece.s_id <> '' THEN
                   #li_StepCase := 40;
               END_IF;

           40:  // write
               "gtyp_Interface_TXT_Controler".Publish.ActionButtonNFCModule.History            := "gtyp_VGR".History;
               "gtyp_Interface_TXT_Controler".Publish.ActionButtonNFCModule.Workpiece.s_type   := "gtyp_VGR".Workpiece.s_type;
               "gtyp_Interface_TXT_Controler".Publish.ActionButtonNFCModule.Workpiece.s_state  := "gtyp_VGR".Workpiece.s_state;

               #li_Return_LDT := RD_SYS_T(#ldt_MQTT);

               "gtyp_Interface_TXT_Controler".Publish.ActionButtonNFCModule.s_cmd  := 'write';
               "gtyp_Interface_TXT_Controler".Publish.ActionButtonNFCModule.ldt_ts := DT_TO_LDT(#ldt_MQTT);

               #li_StepCase := 50;

           50: // wait of answer write 
               #lx_Time_Error := TRUE;
               IF ("gtyp_Interface_TXT_Controler".Subscribe.State_NFC_Device.ldt_ts > "gtyp_Interface_TXT_Controler".Publish.ActionButtonNFCModule.ldt_ts) THEN
                   #lx_Time_Error := FALSE;
                   #li_StepCase := 80;
               END_IF;
               // runtime error
               IF #lfb_TON_Error.Q THEN
                   #lx_Time_Error := FALSE;
                   "gtyp_VGR".x_Workpiece_NiO := TRUE;
                   #li_StepCase := 0;
               END_IF;

           60: // read uid cmd

               #li_Return_LDT := RD_SYS_T(#ldt_MQTT);

               "gtyp_Interface_TXT_Controler".Publish.ActionButtonNFCModule.s_cmd := 'read_uid';
               "gtyp_Interface_TXT_Controler".Publish.ActionButtonNFCModule.ldt_ts := DT_TO_LDT(#ldt_MQTT);
               #lx_Time_Wait   := TRUE;
               #li_StepCase    := 70;

           70: // wait of answer read_uid 
               IF NOT "QX_SSC_LED_Green_Q5" OR #lfb_TON_Wait.Q OR ("gtyp_Interface_TXT_Controler".Subscribe.State_NFC_Device.ldt_ts > "gtyp_Interface_TXT_Controler".Publish.ActionButtonNFCModule.ldt_ts) THEN
                   IF LEN("gtyp_Interface_TXT_Controler".Subscribe.State_NFC_Device.Workpiece.s_id) = 8 THEN
                       "gtyp_Setup".x_Clean_Rack_HBW := TRUE;
                   END_IF;
                   #lx_Time_Wait := FALSE;
                   "gtyp_Interface_TXT_Controler".Subscribe.State_NFC_Device.Workpiece.s_id := '';
                   #li_StepCase := 0;
               END_IF;

           80: // completed

               "gtyp_VGR"."x_NFC_Completed" := TRUE;

               IF NOT "gtyp_VGR".x_NFC_Start AND NOT "gtyp_VGR".x_NFC_Start_First THEN
                   "gtyp_VGR"."x_NFC_Completed" := FALSE;
                   #lx_Start := FALSE;
                   #li_StepCase := 0;
               END_IF;

               // Statement section ELSE
               ELSE  
                   ;
       END_CASE;

   ELSE
       #lx_Init := TRUE;
   END_IF;
END_FUNCTION_BLOCK

FUNCTION_BLOCK "PRG_Acknowledge"   // FB18, SCL
TITLE = Program Acknowledge
{ S7_Optimized_Access := 'TRUE' }
AUTHOR : A.Schaefer
VERSION : 0.0
   VAR
      lx_Init : Bool;
      li_StepCase : Int;
      lldt_Ack_old : LDT;
      lfb_TON_Wait : TON_TIME;
      lx_Start_TON_Wait : Bool;
   END_VAR
BEGIN
   IF #lx_Init THEN
       #lfb_TON_Wait(IN:= #lx_Start_TON_Wait,PT:= T#20s);

       CASE #li_StepCase OF

           0:  // Init
               #lx_Start_TON_Wait := FALSE;

               // check whether acknowledgment has been pressed (time stamp changes)
               IF ("gtyp_Interface_Dashboard".Publish.ldt_AcknowledgeButton > #lldt_Ack_old)
                   OR "gtyp_Setup".x_AcknowledgeButton THEN
                   #lldt_Ack_old    := "gtyp_Interface_Dashboard".Publish.ldt_AcknowledgeButton;
                   #li_StepCase    := 10;
               END_IF;

           10: // acknowledge Errors
               "gtyp_HBW".x_Error := FALSE;
               "gtyp_MPO".x_Error := FALSE;
               "gtyp_SLD".x_Error := FALSE;
               #li_StepCase := 20;

           20: // Reset acknowledge button
               "gtyp_Setup".x_AcknowledgeButton := FALSE;
               #li_StepCase := 0;
       // Statement section ELSE
       ELSE  
           ;
       END_CASE;

   ELSE
       #lx_Init := TRUE;
   END_IF;
END_FUNCTION_BLOCK

FUNCTION_BLOCK "PRG_Order"   // FB20, SCL
TITLE = Program Order
{ S7_Optimized_Access := 'TRUE' }
AUTHOR : A.Schaefer
VERSION : 0.0
   VAR
      lx_Init : Bool;
      li_StepCase : Int;
      lldt_ts_old : LDT;
      ldt_MQTT : Date_And_Time;
      li_Return_LDT : Int;
      lfb_TON_Wait : TON_TIME;
      lx_Start_TON_Wait : Bool;
   END_VAR
BEGIN
   IF #lx_Init THEN
       #lfb_TON_Wait(IN:= #lx_Start_TON_Wait,PT:= T#20s);

       // step chain order
       CASE #li_StepCase OF

           0:  // init
               #lx_Start_TON_Wait := FALSE;
               #li_StepCase := 10;

           10: // check whether order button has been pressed (time stamp changes)
               IF ("gtyp_Interface_Dashboard".Publish.OrderWorkpieceButton.ldt_ts > #lldt_ts_old) THEN
                   #li_Return_LDT := RD_SYS_T(#ldt_MQTT);
                   "gtyp_Interface_Dashboard".Subscribe.State_Order.ldt_ts := DT_TO_LDT(#ldt_MQTT);
                   "gtyp_Interface_Dashboard".Subscribe.State_Order.s_state := 'ORDERED';
                   "gtyp_VGR".s_HBW_Outsource_Typ := "gtyp_Interface_Dashboard".Publish.OrderWorkpieceButton.s_type;
                   "gtyp_Interface_Dashboard".Subscribe.State_Order.s_type := "gtyp_VGR".s_HBW_Outsource_Typ;
                   IF "gtyp_VGR".x_Ready_For_Outsource THEN
                       #lldt_ts_old := "gtyp_Interface_Dashboard".Publish.OrderWorkpieceButton.ldt_ts;
                       "gtyp_VGR".x_HBW_Outsource := TRUE;
                       #li_StepCase := 20;
                   END_IF;
               END_IF;

           20: // delete
               IF "gtyp_VGR".x_HBW_PickedUp OR NOT "gtyp_VGR".x_HBW_Outsource THEN
                   "gtyp_VGR".x_HBW_Outsource := FALSE;
                   "gtyp_VGR".s_HBW_Outsource_Typ := '';
                   #li_StepCase := 0;
               END_IF;

       // Statement section ELSE
       ELSE  
                   ;
       END_CASE;

   ELSE
       #lx_Init    := TRUE;
       #lldt_ts_old:= LDT#1970-01-01-00:00:00;
   END_IF;
END_FUNCTION_BLOCK

// folder: 3.1. VGR

FUNCTION_BLOCK "PRG_VGR_Axis_vertical"   // FB1, SCL
TITLE = Program Axis vertical VGR
{ S7_Optimized_Access := 'TRUE' }
AUTHOR : A.Schaefer
VERSION : 0.0
   VAR
      lx_Init : Bool;
      lfb_vertical_Axis : "FB_Axis";
   END_VAR
BEGIN
   IF #lx_Init THEN

       // FB Axis vertical
       #lfb_vertical_Axis(ini_Axis         := 2,
                   indi_Increment          := "gtyp_VGR".vertical_Axis.di_Increment,
                   inx_Ref_Switch          := "IX_VGR_RefSwitchVerticalAxis_I1",
                   inx_Referencing         := "gtyp_VGR".vertical_Axis.x_Reference,
                   inx_Start_Positioning   := "gtyp_VGR".vertical_Axis.x_Start_Positioning,
                   indi_Target_Position    := "gtyp_VGR".vertical_Axis.di_Target_Position,
                   ini_PWM                 := "gtyp_VGR".vertical_Axis.i_PWM,
                   inouttyp_Config         := "gtyp_VGR".vertical_Axis.Config,
                   inouttyp_Setup          := "gtyp_SetupAxis");

       "QX_VGR_M1_VerticalAxisUp_Q1"       := #lfb_vertical_Axis.outx_Motor_Neg;
       "QX_VGR_M1_VerticalAxisDown_Q2"     := #lfb_vertical_Axis.outx_Motor_Pos;
       "QW_VGR_PWM_Vertical_M1"            := #lfb_vertical_Axis.outi_Motor_PWM;
       "gtyp_VGR".vertical_Axis.di_Actual_Position:= #lfb_vertical_Axis.outdi_Actual_Position;
       "gtyp_VGR".vertical_Axis.x_Referenced      := #lfb_vertical_Axis.outx_Referenced;
       "gtyp_VGR".vertical_Axis.x_Position_Reached:= #lfb_vertical_Axis.outx_Position_Reached;
   ELSE
       #lx_Init := TRUE;
   END_IF;
END_FUNCTION_BLOCK

FUNCTION_BLOCK "PRG_VGR_Axis_horizontal"   // FB4, SCL
TITLE = Program Axis horizontal VGR
{ S7_Optimized_Access := 'TRUE' }
AUTHOR : A.Schaefer
VERSION : 0.0
   VAR
      lx_Init : Bool;
      lfb_horizontal_Axis : "FB_Axis";
   END_VAR
BEGIN
   IF #lx_Init THEN

       // FB Axis horizontal
       #lfb_horizontal_Axis(ini_Axis       := 1,
                   indi_Increment          := "gtyp_VGR".horizontal_Axis.di_Increment,
                   inx_Ref_Switch          := "IX_VGR_RefSwitchHorizontalAxis_I2",
                   inx_Referencing         := "gtyp_VGR".horizontal_Axis.x_Reference,
                   inx_Start_Positioning   := "gtyp_VGR".horizontal_Axis.x_Start_Positioning,
                   indi_Target_Position    := "gtyp_VGR".horizontal_Axis.di_Target_Position,
                   ini_PWM                 := "gtyp_VGR".horizontal_Axis.i_PWM,
                   inouttyp_Config         := "gtyp_VGR".horizontal_Axis.Config,
                   inouttyp_Setup          := "gtyp_SetupAxis");

       "QX_VGR_M2_HorizontalAxisForward_Q4"    := #lfb_horizontal_Axis.outx_Motor_Pos;
       "QX_VGR_M2_HorizontalAxisBackward_Q3"   := #lfb_horizontal_Axis.outx_Motor_Neg;
       "QW_VGR_PWM_Horizontal_M2"              := #lfb_horizontal_Axis.outi_Motor_PWM;
       "gtyp_VGR".horizontal_Axis.di_Actual_Position    := #lfb_horizontal_Axis.outdi_Actual_Position;
       "gtyp_VGR".horizontal_Axis.x_Referenced          := #lfb_horizontal_Axis.outx_Referenced;
       "gtyp_VGR".horizontal_Axis.x_Position_Reached    := #lfb_horizontal_Axis.outx_Position_Reached;
   ELSE
       #lx_Init := TRUE;
   END_IF;
END_FUNCTION_BLOCK

FUNCTION_BLOCK "PRG_VGR_Axis_rotate"   // FB5, SCL
TITLE = Program Axis rotate VGR
{ S7_Optimized_Access := 'TRUE' }
AUTHOR : A.Schaefer
VERSION : 0.0
   VAR
      lx_Init : Bool;
      lfb_rotate_Axis : "FB_Axis";
   END_VAR
BEGIN
   IF #lx_Init THEN

       // FB Axis rotate
       #lfb_rotate_Axis(ini_Axis           := 3,
                   indi_Increment          := "gtyp_VGR".rotate_Axis.di_Increment,
                   inx_Ref_Switch          := "IX_VGR_RefSwitchRotate_I3",
                   inx_Referencing         := "gtyp_VGR".rotate_Axis.x_Reference,
                   inx_Start_Positioning   := "gtyp_VGR".rotate_Axis.x_Start_Positioning,
                   indi_Target_Position    := "gtyp_VGR".rotate_Axis.di_Target_Position,
                   ini_PWM                 := "gtyp_VGR".rotate_Axis.i_PWM,
                   inouttyp_Config         := "gtyp_VGR".rotate_Axis.Config,
                   inouttyp_Setup          := "gtyp_SetupAxis");

       "QX_VGR_M3_RotateClockwise_Q5"          := #lfb_rotate_Axis.outx_Motor_Neg;
       "QX_VGR_M3_RotateCounterclockwise_Q6"   := #lfb_rotate_Axis.outx_Motor_Pos;
       "QW_VGR_PWM_Rotate_M3"                  := #lfb_rotate_Axis.outi_Motor_PWM;
       "gtyp_VGR".rotate_Axis.di_Actual_Position := #lfb_rotate_Axis.outdi_Actual_Position;
       "gtyp_VGR".rotate_Axis.x_Referenced       := #lfb_rotate_Axis.outx_Referenced;
       "gtyp_VGR".rotate_Axis.x_Position_Reached := #lfb_rotate_Axis.outx_Position_Reached;
   ELSE
       #lx_Init := TRUE;
   END_IF;
END_FUNCTION_BLOCK

FUNCTION_BLOCK "PRG_VGR_Ablauf"   // FB7, SCL
TITLE = Program Ablauf VGR
{ S7_Optimized_Access := 'TRUE' }
AUTHOR : A.Schaefer
VERSION : 0.0
   VAR
      lx_Init : Bool;
      lx_Start_TON_Wait : Bool;
      lx_Start_TON_State : Bool;
      lt_TON_Wait : Time;
      ldt_MQTT : Date_And_Time;
      li_Return_LDT : Int;
      li_Lights : Int;
      li_Lights_old : Int;
      lx_State_activ : Bool;
      li_StepCase : Int;
      li_Counter : Int;
      ldi_Pos_SLD_X : DInt;
      ldi_Pos_SLD_Y : DInt;
      ldi_Pos_SLD_Z : DInt;
      ls_Color : String;
      ls_Target : String;
      lfb_TON_Wait : TON_TIME;
      lfb_TON_State : TON_TIME;
      lfb_R_Trig_NiO : R_TRIG;
   END_VAR
BEGIN
   IF #lx_Init THEN

       // Restart after set Positioning
       IF "gtyp_Setup".x_Set_Pos_Activ OR "gtyp_Setup".x_Color_Sensor_Calibration THEN
           #li_StepCase := 0;
       END_IF;

       // wait time state
       #lfb_TON_State(IN := NOT #lx_Start_TON_State,
                       PT := T#2s);

        IF "gtyp_VGR".x_State_Process THEN
            #li_Return_LDT := RD_SYS_T(#ldt_MQTT);
            "gtyp_Interface_Dashboard".Subscribe.State_Order.ldt_ts := DT_TO_LDT(#ldt_MQTT);
        END_IF;

       // state of the robot cyclically transmitted to the cloud
       IF (#lfb_TON_State.Q OR (#li_Lights <> #li_Lights_old)) AND NOT #lx_Start_TON_State THEN
           #li_Lights_old := #li_Lights;
           #lx_Start_TON_State := TRUE;
           #li_Return_LDT := RD_SYS_T(#ldt_MQTT);
           "gtyp_Interface_Dashboard".Subscribe.State_VGR.ldt_ts       := DT_TO_LDT(#ldt_MQTT);
           "gtyp_Interface_Dashboard".Subscribe.State_VGR.i_code       := #li_Lights;
           "gtyp_Interface_Dashboard".Subscribe.State_VGR.s_description:= '';
           "gtyp_Interface_Dashboard".Subscribe.State_VGR.s_station    := 'vgr';
           "gtyp_Interface_Dashboard".Subscribe.State_VGR.s_target     := #ls_Target;
           "gtyp_Interface_Dashboard".Subscribe.State_VGR.x_active     := #lx_State_activ;

           "gtyp_Interface_Dashboard".Subscribe.PosPanTiltUnit.ldt_ts := DT_TO_LDT(#ldt_MQTT);
       END_IF;

       // restart wait time state
       IF NOT #lfb_TON_State.Q AND #lx_Start_TON_State THEN
           #lx_Start_TON_State := FALSE;
       END_IF;

       // rising edge Workpiece NiO
       #lfb_R_Trig_NiO(CLK := "gtyp_VGR".x_Workpiece_NiO);

       IF #lfb_R_Trig_NiO.Q THEN
           #lx_Start_TON_Wait := FALSE;
           #lx_State_activ := FALSE;
           #li_Lights := 4;
           #ls_Target := '';
           "gtyp_VGR".horizontal_Axis.x_Start_Positioning := FALSE;
           "gtyp_VGR".vertical_Axis.x_Start_Positioning := FALSE;
           "gtyp_VGR".rotate_Axis.x_Start_Positioning := FALSE;
           "gtyp_VGR".x_NFC_Start_First := FALSE;
           "gtyp_VGR".x_NFC_Start := FALSE;
           #li_StepCase := 70;
       END_IF;

       // FB TON Wait
       #lfb_TON_Wait(IN := #lx_Start_TON_Wait,
                       PT := #lt_TON_Wait);

       // step chain VGR
       CASE #li_StepCase OF

           0:  // init
               #lx_Start_TON_Wait := FALSE;
               #li_Lights := 1;
               #lx_State_activ := FALSE;
               #ls_Target := '';
               "gtyp_VGR".horizontal_Axis.x_Start_Positioning := FALSE;
               "gtyp_VGR".vertical_Axis.x_Start_Positioning := FALSE;
               "gtyp_VGR".rotate_Axis.x_Start_Positioning := FALSE;
               "gtyp_VGR".x_HBW_Storage := FALSE;
               "gtyp_VGR".x_HBW_Outsource := FALSE;
               "gtyp_VGR".x_NFC_Start_First := FALSE;
               "gtyp_VGR".x_NFC_Start := FALSE;
               "gtyp_VGR".x_Ready_For_Outsource := FALSE;
               "QX_VGR_Compressor_Q7" := FALSE;
               "QX_VGR_ValveVacuum_Q8" := FALSE;

               IF NOT "gtyp_Setup".x_Set_Pos_Activ THEN
                   #li_StepCase := 10;
               END_IF;

           10: // homing vertical axis
               #li_Lights := 2;
               "gtyp_VGR".x_Ready_For_Outsource     := TRUE;
               "gtyp_VGR".vertical_Axis.x_Reference := TRUE;

               IF NOT "gtyp_VGR".vertical_Axis.x_Referenced THEN
                   #li_StepCase := 20;
               END_IF;

           20: // homed vertical axis
               IF "gtyp_VGR".vertical_Axis.x_Referenced THEN
                   "gtyp_VGR".vertical_Axis.x_Reference := FALSE;
                   #li_StepCase := 30;
               END_IF;

           30: // homing horizontal axis
               "gtyp_VGR".horizontal_Axis.x_Reference := TRUE;

               IF NOT "gtyp_VGR".horizontal_Axis.x_Referenced THEN
                   #li_StepCase := 40;
               END_IF;

           40: // homed horizontal axis
               IF "gtyp_VGR".horizontal_Axis.x_Referenced THEN
                   "gtyp_VGR".horizontal_Axis.x_Reference := FALSE;
                   #li_StepCase := 50;
               END_IF;

           50: // homing rotate axis
               "gtyp_VGR".rotate_Axis.x_Reference := TRUE;

               IF NOT "gtyp_VGR".rotate_Axis.x_Referenced THEN
                   #li_StepCase := 60;
               END_IF;

           60: // homed rotate axis
               IF "gtyp_VGR".rotate_Axis.x_Referenced THEN
                   "gtyp_VGR".rotate_Axis.x_Reference := FALSE;
                   #li_StepCase := 70;
               END_IF;

           70: // Deciding which route to take

               #li_Lights := 1;
               #lx_State_activ := FALSE;
               #ls_Target := '';
               "gtyp_VGR".x_Ready_For_Outsource := TRUE;

               // Procedure - bad part
               IF "gtyp_VGR".x_Workpiece_NiO THEN
                   "gtyp_VGR".x_Ready_For_Outsource := FALSE;
                   #li_Lights := 4;
                   #li_StepCase := 1200;
               // Procedure - pick up finished parts blue
               ELSIF NOT "IX_SLD_LightBarrierBlue_I7" THEN
                   #ldi_Pos_SLD_X := "gtyp_VGR".di_Pos_SLD_Blue_horizontal;
                   #ldi_Pos_SLD_Y := "gtyp_VGR".di_Pos_SLD_Blue_vertical;
                   #ldi_Pos_SLD_Z := "gtyp_VGR".di_Pos_SLD_Blue_rotate;
                   "gtyp_VGR".x_Ready_For_Outsource := FALSE;
                   #li_StepCase := 100;
               // Procedure - pick up finished parts red
               ELSIF NOT "IX_SLD_LightBarrierRed_I6" THEN
                   #ldi_Pos_SLD_X := "gtyp_VGR".di_Pos_SLD_Red_horizontal;
                   #ldi_Pos_SLD_Y := "gtyp_VGR".di_Pos_SLD_Red_vertical;
                   #ldi_Pos_SLD_Z := "gtyp_VGR".di_Pos_SLD_Red_rotate;
                   "gtyp_VGR".x_Ready_For_Outsource := FALSE;
                   #li_StepCase := 100;
               // Procedure - pick up finished parts white
               ELSIF NOT "IX_SLD_LightBarrierWhite_I5" THEN
                   #ldi_Pos_SLD_X := "gtyp_VGR".di_Pos_SLD_White_horizontal;
                   #ldi_Pos_SLD_Y := "gtyp_VGR".di_Pos_SLD_White_vertical;
                   #ldi_Pos_SLD_Z := "gtyp_VGR".di_Pos_SLD_White_rotate;
                   "gtyp_VGR".x_Ready_For_Outsource := FALSE;
                   #li_StepCase := 100;
               // Procedure - outsource to manufacturing
               ELSIF "gtyp_VGR".x_HBW_Outsource THEN
                   // Order State
                   "gtyp_Interface_Dashboard".Subscribe.State_Order.ldt_ts := DT_TO_LDT(#ldt_MQTT);
                   "gtyp_Interface_Dashboard".Subscribe.State_Order.s_state := 'ORDERED';
                   "gtyp_Interface_Dashboard".Subscribe.State_Order.s_type := "gtyp_VGR".s_HBW_Outsource_Typ;
                   #li_StepCase := 400;
               // Procedure - store raw parts
               ELSIF NOT "IX_SSC_LightBarrierStorage_I3" THEN
                   "gtyp_VGR".x_Ready_For_Outsource := FALSE;
                   #li_Lights := 2;
                   "gtyp_VGR".x_HBW_Storage  := TRUE;
                   #li_StepCase                := 600;
               END_IF;

           (**************************************************************************************************)
           (****************************    Procedure - pick up finished parts    ****************************)
           (**************************************************************************************************)
           100: // Position of finished part 

               #li_Lights := 2;
               "gtyp_VGR".horizontal_Axis.di_Target_Position := #ldi_Pos_SLD_X;
               "gtyp_VGR".horizontal_Axis.x_Start_Positioning := TRUE;

               "gtyp_VGR".vertical_Axis.x_Reference := TRUE;

               "gtyp_VGR".rotate_Axis.di_Target_Position := #ldi_Pos_SLD_Z;
               "gtyp_VGR".rotate_Axis.x_Start_Positioning := TRUE;

               IF ("gtyp_VGR".horizontal_Axis.di_Actual_Position <= (#ldi_Pos_SLD_X + "gtyp_VGR".horizontal_Axis.Config.di_Pos_Window))
                   AND ("gtyp_VGR".horizontal_Axis.di_Actual_Position >= (#ldi_Pos_SLD_X - "gtyp_VGR".horizontal_Axis.Config.di_Pos_Window))
                   AND "gtyp_VGR".horizontal_Axis.x_Position_Reached THEN
                   "gtyp_VGR".horizontal_Axis.x_Start_Positioning := FALSE;
               END_IF;

               IF ("gtyp_VGR".rotate_Axis.di_Actual_Position <= (#ldi_Pos_SLD_Z + "gtyp_VGR".rotate_Axis.Config.di_Pos_Window))
                   AND ("gtyp_VGR".rotate_Axis.di_Actual_Position >= (#ldi_Pos_SLD_Z - "gtyp_VGR".rotate_Axis.Config.di_Pos_Window))
                   AND "gtyp_VGR".rotate_Axis.x_Position_Reached THEN
                   "gtyp_VGR".rotate_Axis.x_Start_Positioning := FALSE;
               END_IF;

               IF NOT "gtyp_VGR".vertical_Axis.x_Referenced THEN
                   #li_StepCase := 110;
               END_IF;

           110: // position of finished part reached         

               IF ("gtyp_VGR".horizontal_Axis.di_Actual_Position <= (#ldi_Pos_SLD_X + "gtyp_VGR".horizontal_Axis.Config.di_Pos_Window))
                   AND ("gtyp_VGR".horizontal_Axis.di_Actual_Position >= (#ldi_Pos_SLD_X - "gtyp_VGR".horizontal_Axis.Config.di_Pos_Window))
                   AND "gtyp_VGR".horizontal_Axis.x_Position_Reached THEN
                   "gtyp_VGR".horizontal_Axis.x_Start_Positioning := FALSE;
               END_IF;

               IF ("gtyp_VGR".rotate_Axis.di_Actual_Position <= (#ldi_Pos_SLD_Z + "gtyp_VGR".rotate_Axis.Config.di_Pos_Window))
                   AND ("gtyp_VGR".rotate_Axis.di_Actual_Position >= (#ldi_Pos_SLD_Z - "gtyp_VGR".rotate_Axis.Config.di_Pos_Window))
                   AND "gtyp_VGR".rotate_Axis.x_Position_Reached THEN
                   "gtyp_VGR".rotate_Axis.x_Start_Positioning := FALSE;
               END_IF;

               IF "gtyp_VGR".vertical_Axis.x_Referenced THEN
                   "gtyp_VGR".vertical_Axis.x_Reference := FALSE;
               END_IF;

               IF ("gtyp_VGR".horizontal_Axis.di_Actual_Position <= (#ldi_Pos_SLD_X + "gtyp_VGR".horizontal_Axis.Config.di_Pos_Window))
                   AND ("gtyp_VGR".horizontal_Axis.di_Actual_Position >= (#ldi_Pos_SLD_X - "gtyp_VGR".horizontal_Axis.Config.di_Pos_Window))
                   AND "gtyp_VGR".horizontal_Axis.x_Position_Reached
                   AND "gtyp_VGR".vertical_Axis.x_Referenced
                   AND ("gtyp_VGR".rotate_Axis.di_Actual_Position <= (#ldi_Pos_SLD_Z + "gtyp_VGR".rotate_Axis.Config.di_Pos_Window))
                   AND ("gtyp_VGR".rotate_Axis.di_Actual_Position >= (#ldi_Pos_SLD_Z - "gtyp_VGR".rotate_Axis.Config.di_Pos_Window))
                   AND "gtyp_VGR".rotate_Axis.x_Position_Reached THEN
                   "gtyp_VGR".horizontal_Axis.x_Start_Positioning := FALSE;
                   "gtyp_VGR".vertical_Axis.x_Start_Positioning := FALSE;
                   "gtyp_VGR".rotate_Axis.x_Start_Positioning := FALSE;
                   #li_StepCase := 120;
               END_IF;

           120: // wait sequence
               #lx_Start_TON_Wait := TRUE;
               #lt_TON_Wait := T#500ms;

               IF #lfb_TON_Wait.Q THEN
                   #lx_Start_TON_Wait := FALSE;
                   #li_StepCase := 130;
               END_IF;

           130: // Position vertical finished part
               "gtyp_VGR".vertical_Axis.di_Target_Position := #ldi_Pos_SLD_Y;
               "gtyp_VGR".vertical_Axis.x_Start_Positioning := TRUE;

               IF ("gtyp_VGR".vertical_Axis.di_Actual_Position <= (#ldi_Pos_SLD_Y + "gtyp_VGR".vertical_Axis.Config.di_Pos_Window))
                   AND ("gtyp_VGR".vertical_Axis.di_Actual_Position >= (#ldi_Pos_SLD_Y - "gtyp_VGR".vertical_Axis.Config.di_Pos_Window))
                   AND "gtyp_VGR".vertical_Axis.x_Position_Reached THEN
                   "gtyp_VGR".vertical_Axis.x_Start_Positioning := FALSE;
                   #li_StepCase := 140;
               END_IF;

           140: // start compressor
               "QX_VGR_Compressor_Q7" := TRUE;

               #lx_Start_TON_Wait := TRUE;
               #lt_TON_Wait := T#1000ms;

               IF #lfb_TON_Wait.Q THEN
                   #lx_Start_TON_Wait := FALSE;
                   #li_StepCase := 150;
               END_IF;

           150: // turn on the vacuum and pick up the part
               "QX_VGR_ValveVacuum_Q8" := true;

               #lx_Start_TON_Wait := TRUE;
               #lt_TON_Wait := T#1000ms;

               IF #lfb_TON_Wait.Q THEN
                   #lx_Start_TON_Wait := FALSE;
                   #lx_State_activ := TRUE;
                   #ls_Target := 'dso';
                   "gtyp_VGR".History   := "gtyp_SLD".History;
                   "gtyp_VGR".Workpiece := "gtyp_SLD".Workpiece;
                   "gtyp_SLD".Workpiece.s_id := '0';
                   "gtyp_SLD".Workpiece.s_state := '';
                   "gtyp_SLD".Workpiece.s_type := '';
                   FOR #li_Counter := 1 TO 8 DO
                       "gtyp_SLD".History[#li_Counter].i_code := 0;
                       "gtyp_SLD".History[#li_Counter].ldt_ts := DT#1990-01-01-00:00:00;
                   END_FOR;

                   #li_Return_LDT := RD_SYS_T(#ldt_MQTT);
                   "gtyp_VGR".History[8].i_code := 800;
                   "gtyp_VGR".History[8].ldt_ts := DT_TO_LDT(#ldt_MQTT);

                   "gtyp_Interface_Dashboard".Subscribe.State_SLD.x_active := FALSE;

                   #li_StepCase := 160;
               END_IF;

           160: // Position vertical preposition NFC
               "gtyp_VGR".vertical_Axis.di_Target_Position := "gtyp_VGR".di_Pos_NFC_vertical - "gtyp_VGR".di_Offset_Pos_DSI_NFC_vertical;
               "gtyp_VGR".vertical_Axis.x_Start_Positioning := TRUE;

               IF ("gtyp_VGR".vertical_Axis.di_Actual_Position <= ("gtyp_VGR".di_Pos_NFC_vertical - "gtyp_VGR".di_Offset_Pos_DSI_NFC_vertical + "gtyp_VGR".vertical_Axis.Config.di_Pos_Window))
                   AND ("gtyp_VGR".vertical_Axis.di_Actual_Position >= ("gtyp_VGR".di_Pos_NFC_vertical - "gtyp_VGR".di_Offset_Pos_DSI_NFC_vertical - "gtyp_VGR".vertical_Axis.Config.di_Pos_Window))
                   AND "gtyp_VGR".vertical_Axis.x_Position_Reached THEN
                   "gtyp_VGR".vertical_Axis.x_Start_Positioning := FALSE;
                   #li_StepCase := 170;
               END_IF;

           170: // homing horizontal axis
               "gtyp_VGR".horizontal_Axis.x_Reference := TRUE;

               IF NOT "gtyp_VGR".horizontal_Axis.x_Referenced THEN
                   #li_StepCase := 180;
               END_IF;

           180: // homed horizontal axis
               IF "gtyp_VGR".horizontal_Axis.x_Referenced THEN
                   "gtyp_VGR".horizontal_Axis.x_Reference           := FALSE;
                   #li_StepCase := 190;
               END_IF;

           190: // wait sequence
               #lx_Start_TON_Wait := TRUE;
               #lt_TON_Wait := T#500ms;

               IF #lfb_TON_Wait.Q THEN
                   #lx_Start_TON_Wait := FALSE;
                   #li_StepCase := 200;
               END_IF;

           200: // Position horizontal/rotate NFC

               "gtyp_VGR".horizontal_Axis.di_Target_Position := "gtyp_VGR".di_Pos_NFC_horizontal;
               "gtyp_VGR".horizontal_Axis.x_Start_Positioning := TRUE;
               "gtyp_VGR".rotate_Axis.di_Target_Position := "gtyp_VGR".di_Pos_NFC_rotate;
               "gtyp_VGR".rotate_Axis.x_Start_Positioning := TRUE;

               IF ("gtyp_VGR".horizontal_Axis.di_Actual_Position <= ("gtyp_VGR".di_Pos_NFC_horizontal + "gtyp_VGR".horizontal_Axis.Config.di_Pos_Window))
                   AND ("gtyp_VGR".horizontal_Axis.di_Actual_Position >= ("gtyp_VGR".di_Pos_NFC_horizontal - "gtyp_VGR".horizontal_Axis.Config.di_Pos_Window))
                   AND "gtyp_VGR".horizontal_Axis.x_Position_Reached THEN
                   "gtyp_VGR".horizontal_Axis.x_Start_Positioning := FALSE;
               END_IF;

               IF ("gtyp_VGR".rotate_Axis.di_Actual_Position <= ("gtyp_VGR".di_Pos_NFC_rotate + "gtyp_VGR".rotate_Axis.Config.di_Pos_Window))
                   AND ("gtyp_VGR".rotate_Axis.di_Actual_Position >= ("gtyp_VGR".di_Pos_NFC_rotate - "gtyp_VGR".rotate_Axis.Config.di_Pos_Window))
                   AND "gtyp_VGR".rotate_Axis.x_Position_Reached THEN
                   "gtyp_VGR".rotate_Axis.x_Start_Positioning := FALSE;
               END_IF;

               IF ("gtyp_VGR".horizontal_Axis.di_Actual_Position <= ("gtyp_VGR".di_Pos_NFC_horizontal + "gtyp_VGR".horizontal_Axis.Config.di_Pos_Window))
                   AND ("gtyp_VGR".horizontal_Axis.di_Actual_Position >= ("gtyp_VGR".di_Pos_NFC_horizontal - "gtyp_VGR".horizontal_Axis.Config.di_Pos_Window))
                   AND "gtyp_VGR".horizontal_Axis.x_Position_Reached
                   AND ("gtyp_VGR".rotate_Axis.di_Actual_Position <= ("gtyp_VGR".di_Pos_NFC_rotate + "gtyp_VGR".rotate_Axis.Config.di_Pos_Window))
                   AND ("gtyp_VGR".rotate_Axis.di_Actual_Position >= ("gtyp_VGR".di_Pos_NFC_rotate - "gtyp_VGR".rotate_Axis.Config.di_Pos_Window))
                   AND "gtyp_VGR".rotate_Axis.x_Position_Reached THEN
                   "gtyp_VGR".horizontal_Axis.x_Start_Positioning := FALSE;
                   "gtyp_VGR".rotate_Axis.x_Start_Positioning := FALSE;
                   #li_StepCase := 210;
               END_IF;

           210: // wait sequence
               #lx_Start_TON_Wait := TRUE;
               #lt_TON_Wait := T#500ms;

               IF #lfb_TON_Wait.Q THEN
                   #lx_Start_TON_Wait := FALSE;
                   #li_StepCase := 220;
               END_IF;

           220: // Position vertical NFC

               "gtyp_VGR".vertical_Axis.di_Target_Position := "gtyp_VGR".di_Pos_NFC_vertical;
               "gtyp_VGR".vertical_Axis.x_Start_Positioning := TRUE;

               IF ("gtyp_VGR".vertical_Axis.di_Actual_Position <= ("gtyp_VGR".di_Pos_NFC_vertical + "gtyp_VGR".vertical_Axis.Config.di_Pos_Window))
                   AND ("gtyp_VGR".vertical_Axis.di_Actual_Position >= ("gtyp_VGR".di_Pos_NFC_vertical - "gtyp_VGR".vertical_Axis.Config.di_Pos_Window))
                   AND "gtyp_VGR".vertical_Axis.x_Position_Reached THEN
                   "gtyp_VGR".vertical_Axis.x_Start_Positioning := FALSE;
                   #li_StepCase := 230;
               END_IF;

           230: // Start write/read NFC

               "gtyp_VGR".x_NFC_Start := TRUE;

               IF "gtyp_VGR".x_NFC_Completed THEN
                   "gtyp_VGR".x_NFC_Start := FALSE;
                   #li_StepCase := 240;
               END_IF;

           240: // homing vertical axis

               "gtyp_VGR".vertical_Axis.x_Reference := TRUE;

               IF NOT "gtyp_VGR".vertical_Axis.x_Referenced THEN
                   #li_StepCase := 250;
               END_IF;

           250: // homed vertical axis
               IF "gtyp_VGR".vertical_Axis.x_Referenced THEN
                   "gtyp_VGR".vertical_Axis.x_Reference := FALSE;
                   #li_StepCase := 260;
               END_IF;

           260: // wait sequence
               #lx_Start_TON_Wait := TRUE;
               #lt_TON_Wait := T#500ms;

               IF #lfb_TON_Wait.Q THEN
                   #lx_Start_TON_Wait := FALSE;
                   #li_StepCase := 270;
               END_IF;

           270: // Position horizontal/rotate DSO Output

               "gtyp_VGR".horizontal_Axis.di_Target_Position := "gtyp_VGR".di_Pos_DSO_horizontal;
               "gtyp_VGR".horizontal_Axis.x_Start_Positioning := TRUE;

               "gtyp_VGR".rotate_Axis.di_Target_Position := "gtyp_VGR".di_Pos_DSO_rotate;
               "gtyp_VGR".rotate_Axis.x_Start_Positioning := TRUE;

               IF ("gtyp_VGR".horizontal_Axis.di_Actual_Position <= ("gtyp_VGR".di_Pos_DSO_horizontal + "gtyp_VGR".horizontal_Axis.Config.di_Pos_Window))
                   AND ("gtyp_VGR".horizontal_Axis.di_Actual_Position >= ("gtyp_VGR".di_Pos_DSO_horizontal - "gtyp_VGR".horizontal_Axis.Config.di_Pos_Window))
                   AND "gtyp_VGR".horizontal_Axis.x_Position_Reached THEN
                   "gtyp_VGR".horizontal_Axis.x_Start_Positioning := FALSE;
               END_IF;

